# B&R Automation Studio project NAELD004C00R10L518F00 (part 40)

#### Act_Background_TCPSend.st
```iecst
(** 2021-08-01 **)
ACTION Act_Background_TCPSend:

	//Message Send (Generate XML Message)
	IF a_eMsgSend[0] <> HermesMsgTypeNA THEN

		IF a_eMsgSend[0] = HermesMsgTypeCheckAlive THEN
			fHermesFormCheckAlive(ADR(a_tyXMLTableDataSnd) , p_tyDTStructure , tyCheckAliveSnd);
			fTableConvertToXML(ADR(sSnd) , ADR(udiSndMsgLen) , SIZEOF(sSnd) , ADR(a_tyXMLTableDataSnd) , ADR(a_tyXMLTableDataSnd[0].sTitle) , ADR(a_tyXMLTableDataSnd[0].sValue) , ADR(a_tyXMLTableDataSnd[0].uiSize) , SIZEOF(a_tyXMLTableDataSnd[0]) , 12);

		ELSIF a_eMsgSend[0] = HermesMsgTypeCheckAlivePing THEN
			fHermesFormCheckAlive(ADR(a_tyXMLTableDataSnd) , p_tyDTStructure , tyCheckAlivePingSnd);
			fTableConvertToXML(ADR(sSnd) , ADR(udiSndMsgLen) , SIZEOF(sSnd) , ADR(a_tyXMLTableDataSnd) , ADR(a_tyXMLTableDataSnd[0].sTitle) , ADR(a_tyXMLTableDataSnd[0].sValue) , ADR(a_tyXMLTableDataSnd[0].uiSize) , SIZEOF(a_tyXMLTableDataSnd[0]) , 12);

		ELSIF a_eMsgSend[0] = HermesMsgTypeCheckAlivePong THEN
			fHermesFormCheckAlive(ADR(a_tyXMLTableDataSnd) , p_tyDTStructure , tyCheckAlivePongSnd);
			fTableConvertToXML(ADR(sSnd) , ADR(udiSndMsgLen) , SIZEOF(sSnd) , ADR(a_tyXMLTableDataSnd) , ADR(a_tyXMLTableDataSnd[0].sTitle) , ADR(a_tyXMLTableDataSnd[0].sValue) , ADR(a_tyXMLTableDataSnd[0].uiSize) , SIZEOF(a_tyXMLTableDataSnd[0]) , 12);

		ELSIF a_eMsgSend[0] = HermesMsgTypeServiceDescription THEN
			fHermesFormServiceDescription(ADR(a_tyXMLTableDataSnd) , p_tyDTStructure , tyServiceDescriptionSnd);
			fTableConvertToXML(ADR(sSnd) , ADR(udiSndMsgLen) , SIZEOF(sSnd) , ADR(a_tyXMLTableDataSnd) , ADR(a_tyXMLTableDataSnd[0].sTitle) , ADR(a_tyXMLTableDataSnd[0].sValue) , ADR(a_tyXMLTableDataSnd[0].uiSize) , SIZEOF(a_tyXMLTableDataSnd[0]) , 30);

		ELSIF a_eMsgSend[0] = HermesMsgTypeNotification THEN
			fHermesFormNotification(ADR(a_tyXMLTableDataSnd) , p_tyDTStructure , tyNotificationSnd);
			fTableConvertToXML(ADR(sSnd) , ADR(udiSndMsgLen) , SIZEOF(sSnd) , ADR(a_tyXMLTableDataSnd) , ADR(a_tyXMLTableDataSnd[0].sTitle) , ADR(a_tyXMLTableDataSnd[0].sValue) , ADR(a_tyXMLTableDataSnd[0].uiSize) , SIZEOF(a_tyXMLTableDataSnd[0]) , 14);

		ELSIF a_eMsgSend[0] = HermesMsgTypeBoardAvailable THEN
			fHermesFormBoardAvailable(ADR(a_tyXMLTableDataSnd) , p_tyDTStructure , tyBoardAvailableSnd);
			fTableConvertToXML(ADR(sSnd) , ADR(udiSndMsgLen) , SIZEOF(sSnd) , ADR(a_tyXMLTableDataSnd) , ADR(a_tyXMLTableDataSnd[0].sTitle) , ADR(a_tyXMLTableDataSnd[0].sValue) , ADR(a_tyXMLTableDataSnd[0].uiSize) , SIZEOF(a_tyXMLTableDataSnd[0]) , 50);

		ELSIF a_eMsgSend[0] = HermesMsgTypeRevokeBoardAvl THEN
			fHermesFormRevokeBoardAvailable(ADR(a_tyXMLTableDataSnd) , p_tyDTStructure);
			fTableConvertToXML(ADR(sSnd) , ADR(udiSndMsgLen) , SIZEOF(sSnd) , ADR(a_tyXMLTableDataSnd) , ADR(a_tyXMLTableDataSnd[0].sTitle) , ADR(a_tyXMLTableDataSnd[0].sValue) , ADR(a_tyXMLTableDataSnd[0].uiSize) , SIZEOF(a_tyXMLTableDataSnd[0]) , 8);

		ELSIF a_eMsgSend[0] = HermesMsgTypeMachineReady THEN
			eStatus1	:= Error;
			udiStatus1	:= 10135;	//Machine Ready Request To Send From Downstream Hermes

		ELSIF a_eMsgSend[0] = HermesMsgTypeRevokeMachineReady THEN
			eStatus1	:= Error;
			udiStatus1	:= 10136;	//Revoke Machine Ready Request To Send From Downstream Hermes

		ELSIF a_eMsgSend[0] = HermesMsgTypeStartTransport THEN
			eStatus1	:= Error;
			udiStatus1	:= 10137;	//Start Transport Request To Send From Downstream Hermes

		ELSIF a_eMsgSend[0] = HermesMsgTypeStopTransport THEN
			eStatus1	:= Error;
			udiStatus1	:= 10110;	//Stop Transport Request To Send From Downstream Hermes

		ELSIF a_eMsgSend[0] = HermesMsgTypeTransportFinished THEN
			fHermesFormTransportFinished(ADR(a_tyXMLTableDataSnd) , p_tyDTStructure , tyTransportFinished);
			fTableConvertToXML(ADR(sSnd) , ADR(udiSndMsgLen) , SIZEOF(sSnd) , ADR(a_tyXMLTableDataSnd) , ADR(a_tyXMLTableDataSnd[0].sTitle) , ADR(a_tyXMLTableDataSnd[0].sValue) , ADR(a_tyXMLTableDataSnd[0].uiSize) , SIZEOF(a_tyXMLTableDataSnd[0]) , 12);

		ELSIF a_eMsgSend[0] = HermesMsgTypeSetConfiguration THEN
			eStatus1	:= Error;
			udiStatus1	:= 10138;	//Set Configuration Request To Send From Downstream Hermes

		ELSIF a_eMsgSend[0] = HermesMsgTypeGetConfiguration THEN
			eStatus1	:= Error;
			udiStatus1	:= 10139;	//Get Configuration Request To Send From Downstream Hermes

		ELSIF a_eMsgSend[0] = HermesMsgTypeCurrConfiguration THEN
			eStatus1	:= Error;
			udiStatus1	:= 10140;	//Current Configuration Request To Send From Downstream Hermes

		ELSIF a_eMsgSend[0] = HermesMsgTypeBoardForecast THEN
			fHermesFormBoardForecast(ADR(a_tyXMLTableDataSnd) , p_tyDTStructure , tyBoardForecastSnd);
			fTableConvertToXML(ADR(sSnd) , ADR(udiSndMsgLen) , SIZEOF(sSnd) , ADR(a_tyXMLTableDataSnd) , ADR(a_tyXMLTableDataSnd[0].sTitle) , ADR(a_tyXMLTableDataSnd[0].sValue) , ADR(a_tyXMLTableDataSnd[0].uiSize) , SIZEOF(a_tyXMLTableDataSnd[0]) , 50);

		ELSIF a_eMsgSend[0] = HermesMsgTypeQueryBoardInfo THEN
			eStatus1	:= Error;
			udiStatus1	:= 10142;	//Query Board Info Request To Send From Downstream Hermes

		ELSIF a_eMsgSend[0] = HermesMsgTypeSendBoardInfo THEN
			fHermesFormSendBoardInfo(ADR(a_tyXMLTableDataSnd) , p_tyDTStructure , tySendBoardInfo);
			fTableConvertToXML(ADR(sSnd) , ADR(udiSndMsgLen) , SIZEOF(sSnd) , ADR(a_tyXMLTableDataSnd) , ADR(a_tyXMLTableDataSnd[0].sTitle) , ADR(a_tyXMLTableDataSnd[0].sValue) , ADR(a_tyXMLTableDataSnd[0].uiSize) , SIZEOF(a_tyXMLTableDataSnd[0]) , 40);
			bFoundTop	   := FALSE;
			bFoundBottom   := FALSE;
			bFoundNothing  := FALSE;
			bSearchTop     := FALSE;
			bSearchBottom  := FALSE;
			bSendOk        := FALSE;
			tyMsgTypeRcv.bQueryBoardInfo := FALSE;
			//10159

		ELSIF a_eMsgSend[0] = HermesMsgTypeQueryWorkOrderInfo THEN
			eStatus1	:= Error;
			udiStatus1	:= 10160;	//Query Work Order Info Request To Send From Downstream Hermes

		ELSIF a_eMsgSend[0] = HermesMsgTypeSendWorkOrderInfo THEN
			eStatus1	:= Error;
			udiStatus1	:= 10161;	//Send Work Order Info Request To Send From Downstream Hermes

		ELSIF a_eMsgSend[0] = HermesMsgTypeBoardArrived THEN
			eStatus1	:= Error;
			udiStatus1	:= 10162;	//BoardArrived Request To Send From Downstream Hermes

		ELSIF a_eMsgSend[0] = HermesMsgTypeBoardDeparted THEN
			eStatus1	:= Error;
			udiStatus1	:= 10163;	//BoardDeparted Request To Send From Downstream Hermes

		END_IF

		//Message Send
		IF p_bInternalUse = FALSE THEN
			fbSend.udiTCPIdent	:= udiClntIdent;
			fbSend.udiSndSize	:= udiSndMsgLen;
			fbSend(bEn := TRUE);
		ELSE
			sInternalSnd	:= sSnd;
		END_IF

		IF (fbSend.udiStatus = 0) OR (p_bInternalUse = TRUE) THEN

			fLogDTConvert(ADR(sDT) , p_dtCurrDT);
			memset(ADR(a_sLogList[udiLogCntr]) , 0 , SIZEOF(a_sLogList[udiLogCntr]));
			memcpy(ADR(a_sLogList[udiLogCntr]) + LEN(a_sLogList[udiLogCntr]) , ADR(sDT) , LEN(sDT));
			memcpy(ADR(a_sLogList[udiLogCntr]) + LEN(a_sLogList[udiLogCntr]) , ADR('$r$n') , LEN('$r$n'));
			memcpy(ADR(a_sLogList[udiLogCntr]) + LEN(a_sLogList[udiLogCntr]) , ADR('SND_TO_DS$r$n') , LEN('SND_TO_DS$r$n'));
			memcpy(ADR(a_sLogList[udiLogCntr]) + LEN(a_sLogList[udiLogCntr]) , ADR(sSnd) , LEN(sSnd));
			memcpy(ADR(a_sLogList[udiLogCntr]) + LEN(a_sLogList[udiLogCntr]) , ADR('$r$n$r$n') , LEN('$r$n$r$n'));

			udiLogCntr	:= udiLogCntr + 1;
			IF udiLogCntr = 11 THEN
				udiLogCntr	:= 1;
			END_IF

			Act_Background_NotificationSnd;
			fHermesRmvOneMsgSend(ADR(a_eMsgSend) , ADR(udiMsgSendBffr));

			fbSend(bEn := FALSE);

		ELSIF (fbSend.udiStatus = 2321) AND (p_bInternalUse = FALSE) THEN
			bRstConnection	:= TRUE;

		ELSIF (fbSend.udiStatus < 65534) AND (p_bInternalUse = FALSE) THEN
			eStatus1	:= Error;

			IF fbSend.udiStatus = 2300 THEN
				udiStatus1	:= 10143;	//Invalid Ident While Sending Data
			ELSIF fbSend.udiStatus = 2320 THEN
				udiStatus1	:= 10144;	//TCP Retry Send Data Error While Sending Data
			ELSIF fbSend.udiStatus = 2322 THEN
				udiStatus1	:= 10145;	//TCP Send Data Error
			ELSE
				udiStatus1	:= fbSend.udiStatus;
			END_IF

		END_IF

	END_IF

END_ACTION
```

#### Act_InitGlobal.st
```iecst
(** 2019-03-25 **)
ACTION Act_InitGlobal:

	(* Always Change If Project Change *)

	//Pass Data To Link
	p_bLinkStartupRun ACCESS p_StartupRun;
	p_eLinkMcParamDSCommMod ACCESS p_McParamDSCommAMod;

	p_usiLinkProdRcpCurrRcpFlipBrd ACCESS p_ProdRcpCurrRcp2FlippedBrd;
	p_bLinkConvHvBrd ACCESS p_PullConvHvBrd;
	p_bLinkOpsTravLifLDDSComm ACCESS p_OpsTravLifLDDSComm;
	p_eLinkTravLifLDPosGo ACCESS p_OpsTravLifLDPosGo;

	//Pass Data To Internal Use
	p_udiRstErr ACCESS p_RstErrReset;
	p_bPrep ACCESS p_NtParamHermesPrep;
	p_tyParam ACCESS p_HermesDSParam1;
	p_sIPAddr ACCESS p_HWInfoIPAddr;
	pa_usiMacAddr ACCESS p_HWInfoMacAddr;
	p_tyDTStructure ACCESS p_TimeCurrDTStruct;
	p_dtCurrDT ACCESS p_TimeCurrDT;
	p_sMcId ACCESS p_McParamMcNm;
	p_sRecipeNm ACCESS p_ProdRcpCurrRcp1Nm;
	p_sWorkOrderId ACCESS p_AutoRcpWorkOrderId; //from autorcp /////////p_SvyHermesWorkOrderId; //Work Order Id from SupervisoryHermes
	p_sBatchId ACCESS p_SvyHermesBatchId; //Batch Id from SupervisoryHermes
	p_diWidthInUM ACCESS p_ProdRcpCurrRcp1Width;
	p_udiAliveIdleTimeInSec ACCESS p_NtParamDSHermesAAliveTmInSec;
	p_tConnTimeOut ACCESS p_NtParamDSHermesAConnTO;
	p_diTransferInTO ACCESS p_McParamTranOutErrDlyTm;
	pa_tyXMLTableDataBrdAvl ACCESS p_HermesBrdAvlDataTableLastZ; //Last zone Board Data, for B.A
	p_iXMLTableDataBrdAvlTtlIdx ACCESS p_HermesBrdAvlDataTtlIdxLastZ;  //Last zone Board Data, for B.A
	p_bNewBrdAvlFirstZone ACCESS p_HermesBrdAvlDataNewBrdAvl1stZ; //First zone Board Data, for B.F
	p_bNewBrdAvlLastZone ACCESS p_HermesBrdAvlDataNewBrdAvlLastZ; //Last zone Board Data, for B.A
	p_bOpsRun ACCESS p_OpsRun;
	p_bInterruptSen ACCESS p_DIConvRgtSen; //Last Zone Sensor that give B.A
	p_udiFileKeepDay ACCESS p_NtParamDSHermesAFileKeepDay;
	p_sRetainFileName ACCESS p_NtParamDSHermesRetainFileNm;
	p_sProgNm ACCESS p_NtParamDSHermesAProgNm;
	p_bNtSettingsLoadDone ACCESS p_StartupNtSettingsLoadDone;
	p_bRmtPrep ACCESS p_NtParamHermesRmtPrep;
	p_bRmtEn ACCESS p_McParamHermesRmtEn;
	p_bSvyPrep ACCESS p_NtParamHermesSvyPrep;
	p_bSvyEn ACCESS p_McParamHermesSvyEn;
	p_bOpsGConv1HvBrd ACCESS p_PullConvHvBrd; //Take Zone 1's Have Board
	//p_tyUSBoardArrivedData ACCESS p_USHermesBoardArrivedData;
	//p_rAWCycleTm ACCESS p_NtParamDSHermesAWCycleTm;
	p_bInitDone ACCESS p_OpsTravLifLDInitDone;
	p_bFirstZoneEndSen ACCESS p_DIConvRgtSen; //Take First Zone's End sensor
	p_tyHermesConfiguration ACCESS p_HermesConfiguration;
//	p_bUSHermesStopTransport ACCESS p_USHermesStopTransportSnd;
//	p_bRcvBoardInfo ACCESS p_USHermesRcvBoardInfoOk;
//	p_tyBoardInfoData ACCESS p_USHermesBoardInfoData; //SendBoardInfo from Upstream, used to generate B.A for inserted PCB
//	p_bUSHermesTransporting ACCESS p_USHermesTransporting;
	p_eLinkCustomerReq ACCESS p_NtParamCustomerReq;
	p_usiProdRcpCurrRcp1McMod  ACCESS  p_ProdRcpCurrRcp1McMod;      //ADD
//	p_usiSelProdRcpStep  ACCESS p_SelProdRcpStep;

	// phase 1
	p_tySendWorkOrderData ACCESS p_SvyHermesSendWorkOrderData;
	p_bReplyWorkOrderInfo ACCESS  p_ReplyWorkOrderInfo;
	p_bSendBoardForecast ACCESS p_SendBoardForecast;
	p_bClearWorkOrder ACCESS p_ClearWorkOrder;

	p_tyAutoRcpTravLif ACCESS p_AutoRcpTravLif;
	p_diLinkAutoRcpTravLifWidth ACCESS p_AutoRcpTravLifWidth;
	p_diLinkAutoRcpMag1Width ACCESS p_diAutoRcpMag1Width;
	p_diLinkAutoRcpMag2Width ACCESS p_diAutoRcpMag2Width;
	p_diLinkAutoRcpMag3Width ACCESS p_diAutoRcpMag3Width;

	p_tyAutoRcpMagRcp ACCESS p_AutoRcpMagRcp;
	p_ausiSvyMagAccOrder ACCESS p_SvyHermesMagAccOrder;

	p_sHermesBrdId ACCESS p_HermesBrdId;
	p_bDIPullerRetRS ACCESS p_DIPullerRetRS;
	(* Always Change If Project Change *)
END_ACTION
```

#### Act_Initial.st
```iecst
(** 2021-08-01 **)
ACTION Act_Initial:

	//Initial
	sStatTxt	:= a_sStatText[eStat];

	fbCreateSvr.udiSndBffrSize		:= p_udiSndBffrSize;
	fbCreateSvr.udiRcvBffrSize		:= p_udiRcvBffrSize;
	fbCreateSvr.udiAliveIdleTmInSec	:= p_udiAliveIdleTimeInSec;
	fbCreateSvr(bEn := FALSE);

	fbListen(bEn := FALSE);

	fbRcv.udiBffrSize	:= SIZEOF(sRcv);
	fbRcv.p_BffrDest	:= ADR(sRcv);
	fbRcv(bEn := FALSE);

	fbSend.p_BffrDest	:= ADR(sSnd);
	fbSend(bEn := FALSE);

	fbCloseSvr(bEn := FALSE);
	fbCloseClnt(bEn := FALSE);

	fbParseXMLTable.p_XMLTable	:= ADR(a_tyXMLTableDataRcv);

	fbCheckAlive(bEn := FALSE);

	fbCheckAliveSendPing(bEn := FALSE);

	fbCheckAliveRcvPing(bEn := FALSE);

	fbSequenceDS.p_tyMsgTypeRcv	:= ADR(tyMsgTypeRcv);
	fbSequenceDS(bEn := FALSE);

	fbSequenceTO(bEn := FALSE);

	fbFileAppend1.sDevice	:= 'Log';
	fbFileAppend1(bEn := FALSE);

	fbFileOldDel1.sDevice			:= 'Log';
	fbFileOldDel1.sPath				:= '';
	fbFileOldDel1.sKeyword			:= p_sProgNm;
	fbFileOldDel1.udiFileKeepDay	:= p_udiFileKeepDay;
	fbFileOldDel1(bEn := FALSE);

	fbFileRead1.sDevice			:= 'Retain';
	fbFileRead1.sFile			:= p_sRetainFileName;
	fbFileRead1.udiOffset		:= 0;
	fbFileRead1(bEn := FALSE);

	fbFileWrite1.sDevice		:= 'Retain';
	fbFileWrite1.sFile			:= p_sRetainFileName;
	fbFileWrite1.udiOffset		:= 0;
	fbFileWrite1.udiOption		:= 0;
	fbFileWrite1(bEn := FALSE);

END_ACTION
```

#### Act_InitLocal.st
```iecst
(** 2021-08-01 **)
ACTION Act_InitLocal:

	//Input Reference Link To Local Variable
	p_eAct ACCESS ADR(eAct);
	p_udiRstErr ACCESS ADR(udiRstErr);
	p_bPrep ACCESS ADR(bPrep);
	p_bEn ACCESS ADR(bEn);
	p_bDis ACCESS ADR(bDis);
	p_tyParam ACCESS ADR(tyParam);
	p_sIPAddr ACCESS ADR(sIPAddr);
	pa_usiMacAddr ACCESS ADR(a_usiMacAddr);
	p_tyDTStructure ACCESS ADR(tyDTStructure);
	p_dtCurrDT ACCESS ADR(dtCurrDT);
	p_bRdySnd ACCESS ADR(bRdySnd);
	p_bSndCompl ACCESS ADR(bSndCompl);
	p_bSndIncompl ACCESS ADR(bSndInCompl);
	p_bSndNotStart ACCESS ADR(bSndNotStart);
	p_bBAWidthEn ACCESS ADR(bBAWidthEn);
	p_bBASltEn ACCESS ADR(bBASltEn);
	p_bBFWidthEn ACCESS ADR(bBFWidthEn);
	p_bBFSltEn ACCESS ADR(bBFSltEn);
	p_sForecastId ACCESS ADR(sForecastId);
	p_sBoardId ACCESS ADR(sBoardId);
	p_sMcId ACCESS ADR(sMcId);
	p_sInterfaceId ACCESS ADR(sInterfaceId);
	p_sVersion ACCESS ADR(sVersion);
	p_eFailedBoard ACCESS ADR(eFailedBoard);
	p_sRecipeNm ACCESS ADR(sRecipeNm);
	p_eFlippedBoard ACCESS ADR(eFlippedBoard);
	p_sTopBarcode ACCESS ADR(sTopBarcode);
	p_sBottomBarcode ACCESS ADR(sBottomBarcode);
	p_rLength ACCESS ADR(rLength);
	p_rThickness ACCESS ADR(rThickness);
	p_rConveyorSpeed ACCESS ADR(rConveyorSpeed);
	p_rTopClearanceHeight ACCESS ADR(rTopClearanceHeight);
	p_rBottomClearanceHeight ACCESS ADR(rBottomClearanceHeight);
	p_rWeight ACCESS ADR(rWeight);
	p_sWorkOrderId ACCESS ADR(sWorkOrderId);
	p_sBatchId ACCESS ADR(sBatchId);
	p_diWidthInUM ACCESS ADR(diWidthInUM);
	p_diMinSltValue ACCESS ADR(diMinSltValue);
	p_diMaxSltValue ACCESS ADR(diMaxSltValue);
	p_diPitch ACCESS ADR(diPitch);
	p_diTtlSlt ACCESS ADR(diTtlSlt);
	p_diSltToSltInUM ACCESS ADR(diSltToSltInUM);
	p_udiSndBffrSize ACCESS ADR(udiSndBffrSize);
	p_udiRcvBffrSize ACCESS ADR(udiRcvBffrSize);
	p_udiAliveIdleTimeInSec ACCESS ADR(udiAliveIdleTimeInSec);
	p_tConnTimeOut ACCESS ADR(tConnTimeOut);
	p_diTransferInTO ACCESS ADR(diTransferInTO);
	pa_tyXMLTableDataBrdAvl ACCESS ADR(a_tyXMLTableDataBrdAvl);
	p_iXMLTableDataBrdAvlTtlIdx ACCESS ADR(iXMLTableDataBrdAvlTtlIdx);
	p_bNewBrdAvlFirstZone ACCESS ADR(bNewBrdAvl1);
	p_bNewBrdAvlLastZone ACCESS ADR(bNewBrdAvl2);
	p_bOpsRun ACCESS ADR(bOpsRun);
	p_bInterruptSen ACCESS ADR(bInterruptSen);
	p_udiFileKeepDay ACCESS ADR(udiFileKeepDay);
	p_sRetainFileName ACCESS ADR(sRetainFileName);
	p_udiRetainDataAddr ACCESS ADR(udiRetainDataAddr);
	p_udiRetainDataLen ACCESS ADR(udiRetainDataLen);
	p_sProgNm ACCESS ADR(sProgNm);
	p_bNtSettingsLoadDone ACCESS ADR(bNtSettingsLoadDone);
	p_bRmtPrep ACCESS ADR(bRmtPrep);
	p_bRmtEn ACCESS ADR(bRmtEn);
	p_bSvyPrep ACCESS ADR(bSvyPrep);
	p_bSvyEn ACCESS ADR(bSvyEn);
	p_bOpsGConv1HvBrd ACCESS ADR(bOpsGConv1HvBrd);
	p_tyUSBoardArrivedData ACCESS ADR(tyUSBoardArrivedData);
	p_rMcCycleTm ACCESS ADR(rMachineCycleTime);
	p_rAWCycleTm ACCESS ADR(rAutoWidthCycleTime);
	p_bInitDone ACCESS ADR(bInitDone);
	p_bFirstZoneEndSen ACCESS ADR(bFirstZoneEndSen);
	p_bFirstZoneHaveBoard ACCESS ADR(bFirstZoneHaveBoard);
	p_bNewProduct ACCESS ADR(bNewProduct);
	p_bNewWidth ACCESS ADR(bNewWidth);
	p_tyHermesConfiguration ACCESS ADR(tyHermesCurrConfiguration);
	p_bUSHermesStopTransport ACCESS ADR(bUSHermesStopTransport);
	p_bRcvBoardInfo ACCESS ADR(bRcvBoardInfo);
	p_tyBoardInfoData ACCESS ADR(tyBoardInfoData);
	p_bUSHermesTransporting ACCESS ADR(bUSHermesTransporting);
	p_bInternalUse ACCESS ADR(bInternalUse);
	p_sInternalRcv ACCESS ADR(sInternalRcv);

END_ACTION
```

#### Act_Link.st
```iecst
(** 2021-08-01 **)
ACTION Act_Link:

	//Receive Alive Time
	p_tyParam.tRcvAlive	:= p_tyParam.tSndAlive * 2;

	//Ready Send
	//Transfer Finished
//	IF (p_eLinkConvDir = ConvDirLToR) OR (p_eLinkConvDir = ConvDirRToR) THEN
		IF EDGENEG(p_bFirstZoneEndSen) THEN
			p_bSndCompl	:= TRUE;
		END_IF
//	ELSE
//		IF EDGENEG(p_bLinkDILeftSen) THEN
//			p_bSndCompl	:= TRUE;
//		END_IF
//	END_IF

	//Good Bad Board
//	IF p_bLinkOpsConvGdBrd = TRUE THEN
		p_eFailedBoard	:= HermesGoodBoard;
//	ELSE
//		p_eFailedBoard	:= HermesFailedBoard;
//	END_IF

	//New Product for Board Forecast(Id)
	//p_bNewProduct will be True only when machine accepted new recipe, can perform ChangeOver, i.e Machine Free (all zones).
		//siemen
	IF p_ausiSvyMagAccOrder[1] = 10 AND p_bDIPullerRetRS THEN
		p_bNewProduct := (p_tyAutoRcpTravLif.sWorkOrderId <> p_tyAutoRcpMagRcp[1].sWorkOrderId OR
						p_tyAutoRcpTravLif.sProductTypeId <> p_tyAutoRcpMagRcp[1].sProductTypeId OR
						p_tyAutoRcpTravLif.sBatchId <> p_tyAutoRcpMagRcp[1].sBatchId OR
						p_tyAutoRcpTravLif.rWidth <> p_tyAutoRcpMagRcp[1].rWidth) AND (p_bLinkStartupRun = FALSE);
	ELSIF p_ausiSvyMagAccOrder[2] = 10 AND p_bDIPullerRetRS THEN
		p_bNewProduct := (p_tyAutoRcpTravLif.sWorkOrderId <> p_tyAutoRcpMagRcp[2].sWorkOrderId OR
						p_tyAutoRcpTravLif.sProductTypeId <> p_tyAutoRcpMagRcp[2].sProductTypeId OR
						p_tyAutoRcpTravLif.sBatchId <> p_tyAutoRcpMagRcp[2].sBatchId OR
						p_tyAutoRcpTravLif.rWidth <> p_tyAutoRcpMagRcp[2].rWidth) AND (p_bLinkStartupRun = FALSE);
	ELSIF p_ausiSvyMagAccOrder[3] = 10 AND p_bDIPullerRetRS THEN
		p_bNewProduct := (p_tyAutoRcpTravLif.sWorkOrderId <> p_tyAutoRcpMagRcp[3].sWorkOrderId OR
						p_tyAutoRcpTravLif.sProductTypeId <> p_tyAutoRcpMagRcp[3].sProductTypeId OR
						p_tyAutoRcpTravLif.sBatchId <> p_tyAutoRcpMagRcp[3].sBatchId OR
						p_tyAutoRcpTravLif.rWidth <> p_tyAutoRcpMagRcp[3].rWidth) AND (p_bLinkStartupRun = FALSE);
	ELSE
		p_bNewProduct := FALSE;
	END_IF

	//p_bNewProduct := ((*(EDGEPOS(p_bLinkProdRcpCurrAll[0].sRcpNm = p_bLinkProdRcpCurrAll[1].sRcpNm)*)) AND (p_bLinkStartupRun = FALSE));
	bBFAccNewWidth[1] :=  p_diLinkAutoRcpTravLifWidth = p_diLinkAutoRcpMag1Width AND p_eLinkTravLifLDPosGo = TravLifLDPosUS1;
	bBFAccNewWidth[2] :=	p_diLinkAutoRcpTravLifWidth = p_diLinkAutoRcpMag2Width AND p_eLinkTravLifLDPosGo = TravLifLDPosUS2;
	bBFAccNewWidth[3] :=	p_diLinkAutoRcpTravLifWidth = p_diLinkAutoRcpMag3Width AND p_eLinkTravLifLDPosGo = TravLifLDPosUS3;
	//p_bNewWidth will be True only when machine accepted new width, can perform ChangeOver, i.e Machine Free (all zones).
	//p_bNewWidth :=   (EDGEPOS(bBFAccNewWidth[1]) OR EDGEPOS(bBFAccNewWidth[2]) OR EDGEPOS(bBFAccNewWidth[3])) AND (p_bLinkStartupRun = FALSE);

	p_bRdySnd	:= p_bLinkOpsTravLifLDDSComm AND p_eLinkTravLifLDPosGo = TravLifLDPosDS1;  //DBA

	//Machine Cycle Time
	p_rMcCycleTm ACCESS p_NtParamDSHermesMcCycleTm; //Change this if machine got Worst/Least/Different Cycle Time accordingly

	//Flipped Board
	p_eFlippedBoard	:= USINT_TO_UDINT(p_usiLinkProdRcpCurrRcpFlipBrd);

	//Machine All Empty(for ChangeOver), adjust accordingly                                                            //Add
	bAllZonesEmpty := p_bOpsGConv1HvBrd = FALSE AND p_bFirstZoneEndSen = FALSE;// AND p_bLinkDIPresentSen = FALSE (*AND p_tyDI.bTopCoverSWSig = TRUE*);

	//Machine First Zone have board
	p_bFirstZoneHaveBoard := (p_bUSHermesStopTransport AND p_bOpsGConv1HvBrd) OR (p_bOpsGConv1HvBrd AND p_bUSHermesTransporting = FALSE); //Zone 1 have board, either PCB_In from upstream Or Manually load PCB at Zone 1

END_ACTION
```

#### Act_LinkAction.st
```iecst
(** 2021-08-01 **)
ACTION Act_LinkAction:

	IF p_bLinkStartupRun = TRUE THEN
		p_eAct ACCESS p_StartupDSHermesAAct;
	ELSE
		p_eAct ACCESS ADR(eAct);

		IF EDGEPOS(p_eLinkMcParamDSCommMod = McSetCommModHermes) THEN
			bHermesRun	:= TRUE;
			bHermesStop	:= FALSE;
		END_IF

		IF EDGENEG(p_eLinkMcParamDSCommMod = McSetCommModHermes) THEN
			bHermesRun	:= FALSE;
			bHermesStop	:= TRUE;
		END_IF

		IF bHermesRun = TRUE THEN
			p_eAct	:= HermesActBGStartRun;

			IF (eStat = HermesActBGStartRun) AND (eStatus = Done) THEN
				p_eAct		:= HermesActIdle;
				bHermesRun	:= FALSE;
			END_IF
		END_IF

		IF bHermesStop = TRUE THEN
			p_eAct	:= HermesActBGStopRun;

			IF (eStat = HermesActBGStopRun) AND (eStatus = Done) THEN
				p_eAct		:= HermesActIdle;
				bHermesStop	:= FALSE;
			END_IF
		END_IF

	END_IF

//Delete Old Log File for 24 hours After Machine is Continuous Running 30 Days.

	fbDlyTmr(IN := TRUE);
	IF fbDlyTmr.Q THEN
		fbDeleteLogTmr (IN := TRUE);
		IF fbDeleteLogTmr.Q AND eStatus <> Busy THEN
			p_eAct := HermesActDeleteOldLog;
			IF eStat = HermesActDeleteOldLog AND eStatus = Done THEN
				p_eAct := HermesActIdle;
				fbDlyTmr (IN := FALSE);
				fbDeleteLogTmr (IN := FALSE);
			END_IF
		END_IF
	END_IF
END_ACTION
```

#### Cyclic.st
```iecst
(** 2021-08-01 **)
PROGRAM _CYCLIC

	IF bInitDone = FALSE THEN
		bInitDone	:= TRUE;

		Act_InitLocal;
		Act_InitGlobal;

	ELSIF bInitialDone = FALSE THEN
		IF p_bNtSettingsLoadDone = TRUE THEN
			bInitialDone	:= TRUE;

			Act_Initial;
		END_IF

	ELSE

		Act_RstErr;
		Act_LinkAction;
		Act_Action;
		Act_LinkEn;

		IF (p_bPrep = TRUE) AND (p_bEn = TRUE) AND (p_bDis = FALSE) THEN
			Act_Link;
			Act_Main;
			Act_Background;
			Act_Background_ProcessData;
		ELSE
			Act_Main_Disable;

			IF eStat <> HermesActIdle THEN
				eStatus	:= Done;
			ELSE
				eStatus	:= Idle;
			END_IF
		END_IF

		Act_CombineErr;
		Act_Alarm;
		Act_Alarm1;
		Act_Alarm2;
		Act_Alarm3;
		Act_Alarm4;
	END_IF

END_PROGRAM
```

#### Init.st
```iecst
(** 2021-08-01 **)
PROGRAM _INIT

	(* Always Change If Project Change *)

	//Pass Address To Global Address For External Use
	//Action, State & Status
	p_DSHermesAStat	    	:= ADR(eStat);
	p_DSHermesAStatus    	:= ADR(eMainStatus);
	p_DSHermesAStatTxt    	:= ADR(sStatTxt);

	//Alarm
	p_DSHermesAAlmData    	:= ADR(tyAlmData);
	p_DSHermesAAlmData1	    := ADR(tyAlmData1);
	p_DSHermesAAlmData2    	:= ADR(tyAlmData2);
	p_DSHermesAAlmData3    	:= ADR(tyAlmData3);
	p_DSHermesAAlmData4    	:= ADR(tyAlmData4);//add

	//Output
	p_DSHermesAFileNotFound		    := ADR(bFileNotFound);
	p_DSHermesAConnected		    := ADR(bConnected);
	p_DSHermesAHandshakeDone	    := ADR(bHandshakeDone);
	p_DSHermesAUSRdy			    := ADR(bUSRdy);
	p_DSHermesADSRdy			    := ADR(bDSRdy);
	p_DSHermesAUSGdRdy		    	:= ADR(bUSGdRdy);
	p_DSHermesADSGdRdy		    	:= ADR(bDSGdRdy);
	p_DSHermesATransporting	    	:= ADR(bTransporting);
	p_DSHermesAStopTransport	    := ADR(bStopTransport);
	p_DSHermesAInternalSnd	    	:= ADR(sInternalSnd);
	p_DSHermesATransportFinishedSnd  := ADR(bTransportFinishedSnd);
	p_DSHermesABoardDepartedData     := ADR(tyBoardDepartedInfo);
	p_DSHermesAAllZonesEmpty         := ADR(bAllZonesEmpty);

	p_SendBFId                     := ADR (bSendBFId);        //ADD

	(* Always Change If Project Change *)

END_PROGRAM
```

### DSHermesB.var - Change By Project
```iecst
(*2021-08-01*)
(**)
(*Action & State & Status*)
VAR
	p_DSHermesBStat : UDINT;
	p_DSHermesBStatus : UDINT;
	p_DSHermesBStatTxt : UDINT;
END_VAR
(**)
(*Alarm*)
VAR
	p_DSHermesBAlmData : UDINT;
	p_DSHermesBAlmData1 : UDINT;
	p_DSHermesBAlmData2 : UDINT;
	p_DSHermesBAlmData3 : UDINT;
	p_DSHermesBAlmData4 : UDINT;
END_VAR
(**)
(*Output*)
VAR
	p_DSHermesBFileNotFound : UDINT;
	p_DSHermesBConnected : UDINT;
	p_DSHermesBHandshakeDone : UDINT;
	p_DSHermesBUSRdy : UDINT;
	p_DSHermesBDSRdy : UDINT;
	p_DSHermesBUSGdRdy : UDINT;
	p_DSHermesBDSGdRdy : UDINT;
	p_DSHermesBTransporting : UDINT;
	p_DSHermesBStopTransport : UDINT;
	p_DSHermesBInternalSnd : UDINT;
	p_DSHermesBTransportFinishedSnd : UDINT;
	p_DSHermesBBoardDepartedData : UDINT;
	p_DSHermesBAllZonesEmpty : UDINT;
	p_SendBFIdB : UDINT;
END_VAR
```

### Program Logical/Hermes/DSHermesB (IEC, version 1.00.0) - 1.00.0 - NtHermes v5.00.0 , NtTCP v5.00.0 , NtMessage v5.00.0

#### Init.st - Change By Project
```iecst
(** 2021-08-01 **)
PROGRAM _INIT

	(* Always Change If Project Change *)

	//Pass Address To Global Address For External Use
	//Action, State & Status
	p_DSHermesBStat	    	:= ADR(eStat);
	p_DSHermesBStatus    	:= ADR(eMainStatus);
	p_DSHermesBStatTxt    	:= ADR(sStatTxt);

	//Alarm
	p_DSHermesBAlmData    	:= ADR(tyAlmData);
	p_DSHermesBAlmData1	    := ADR(tyAlmData1);
	p_DSHermesBAlmData2    	:= ADR(tyAlmData2);
	p_DSHermesBAlmData3    	:= ADR(tyAlmData3);
	p_DSHermesBAlmData4    	:= ADR(tyAlmData4);//add

	//Output
	p_DSHermesBFileNotFound		    := ADR(bFileNotFound);
	p_DSHermesBConnected		    	:= ADR(bConnected);
	p_DSHermesBHandshakeDone	    	:= ADR(bHandshakeDone);
	p_DSHermesBUSRdy			    	:= ADR(bUSRdy);
	p_DSHermesBDSRdy			    	:= ADR(bDSRdy);
	p_DSHermesBUSGdRdy		    	:= ADR(bUSGdRdy);
	p_DSHermesBDSGdRdy		    	:= ADR(bDSGdRdy);
	p_DSHermesBTransporting	    	:= ADR(bTransporting);
	p_DSHermesBStopTransport	    	:= ADR(bStopTransport);
	p_DSHermesBInternalSnd	    	:= ADR(sInternalSnd);
	p_DSHermesBTransportFinishedSnd  := ADR(bTransportFinishedSnd);
	p_DSHermesBBoardDepartedData     := ADR(tyBoardDepartedInfo);
	p_DSHermesBAllZonesEmpty         := ADR(bAllZonesEmpty);

	p_SendBFIdB                     := ADR (bSendBFId);        //ADD

	(* Always Change If Project Change *)

END_PROGRAM
```

#### Act_InitGlobal.st - Change By Project
```iecst
(** 2019-03-25 **)
ACTION Act_InitGlobal:

	(* Always Change If Project Change *)

	//Pass Data To Link
	p_bLinkStartupRun ACCESS p_StartupRun;
	p_eLinkMcParamDSCommMod ACCESS p_McParamDSCommBMod;
	p_bLinkNtParamProjLaneBPrep ACCESS p_NtParamProjLaneBPrep;

	p_usiLinkProdRcpCurrRcpFlipBrd ACCESS p_ProdRcpCurrRcp2FlippedBrd;
	p_bLinkConvHvBrd ACCESS p_PullConvHvBrd;
	p_bLinkOpsTravLifLDDSComm ACCESS p_OpsTravLifLDDSComm;
	p_eLinkTravLifLDPosGo ACCESS p_OpsTravLifLDPosGo;

	//Pass Data To Internal Use
	p_udiRstErr ACCESS p_RstErrReset;
	p_bPrep ACCESS p_NtParamHermesPrep;
	p_tyParam ACCESS p_HermesDSParam2;
	p_sIPAddr ACCESS p_HWInfoIPAddr;
	pa_usiMacAddr ACCESS p_HWInfoMacAddr;
	p_tyDTStructure ACCESS p_TimeCurrDTStruct;
	p_dtCurrDT ACCESS p_TimeCurrDT;
	p_sMcId ACCESS p_McParamMcNm;
	p_sRecipeNm ACCESS p_ProdRcpCurrRcp1Nm;
	p_sWorkOrderId ACCESS p_SvyHermesWorkOrderId; //Work Order Id from SupervisoryHermes
	p_sBatchId ACCESS p_SvyHermesBatchId; //Batch Id from SupervisoryHermes
	p_diWidthInUM ACCESS p_ProdRcpCurrRcp1Width;
	p_udiAliveIdleTimeInSec ACCESS p_NtParamDSHermesBAliveTmInSec;
	p_tConnTimeOut ACCESS p_NtParamDSHermesBConnTO;
	p_diTransferInTO ACCESS p_McParamTranOutErrDlyTm;
	pa_tyXMLTableDataBrdAvl ACCESS p_HermesBrdAvlDataTableLastZ; //Last zone Board Data, for B.A
	p_iXMLTableDataBrdAvlTtlIdx ACCESS p_HermesBrdAvlDataTtlIdxLastZ;  //Last zone Board Data, for B.A
	p_bNewBrdAvlFirstZone ACCESS p_HermesBrdAvlDataNewBrdAvl1stZ; //First zone Board Data, for B.F
	p_bNewBrdAvlLastZone ACCESS p_HermesBrdAvlDataNewBrdAvlLastZ; //Last zone Board Data, for B.A
	p_bOpsRun ACCESS p_OpsRun;
	p_bInterruptSen ACCESS p_DIConvRgtSen; //Last Zone Sensor that give B.A
	p_udiFileKeepDay ACCESS p_NtParamDSHermesBFileKeepDay;
	p_sRetainFileName ACCESS p_NtParamDSHermesRetainFileNm;
	p_sProgNm ACCESS p_NtParamDSHermesBProgNm;
	p_bNtSettingsLoadDone ACCESS p_StartupNtSettingsLoadDone;
	p_bRmtPrep ACCESS p_NtParamHermesRmtPrep;
	p_bRmtEn ACCESS p_McParamHermesRmtEn;
	p_bSvyPrep ACCESS p_NtParamHermesSvyPrep;
	p_bSvyEn ACCESS p_McParamHermesSvyEn;
	p_bOpsGConv1HvBrd ACCESS p_PullConvHvBrd; //Take Zone 1's Have Board
//	p_tyUSBoardArrivedData ACCESS p_USHermesBoardArrivedData;
//	p_rAWCycleTm ACCESS p_NtParamDSHermesAWCycleTm;
	p_bInitDone ACCESS p_OpsTravLifLDInitDone;
	p_bFirstZoneEndSen ACCESS p_DIConvRgtSen; //Take First Zone's End sensor
	p_tyHermesConfiguration ACCESS p_HermesConfiguration;
//	p_bUSHermesStopTransport ACCESS p_USHermesStopTransportSnd;
//	p_bRcvBoardInfo ACCESS p_USHermesRcvBoardInfoOk;
//	p_tyBoardInfoData ACCESS p_USHermesBoardInfoData; //SendBoardInfo from Upstream, used to generate B.A for inserted PCB
//	p_bUSHermesTransporting ACCESS p_USHermesTransporting;
	p_eLinkCustomerReq ACCESS p_NtParamCustomerReq;
	p_usiProdRcpCurrRcp1McMod  ACCESS  p_ProdRcpCurrRcp1McMod;      //ADD
//	p_usiSelProdRcpStep  ACCESS p_SelProdRcpStep;

	// phase 1
	p_tySendWorkOrderData ACCESS p_SvyHermesSendWorkOrderData;
	p_bReplyWorkOrderInfo ACCESS  p_ReplyWorkOrderInfo;
	p_bSendBoardForecast ACCESS p_SendBoardForecast;
	p_bClearWorkOrder ACCESS p_ClearWorkOrder;

	(* Always Change If Project Change *)
END_ACTION
```

#### InputRef_Link.var - Change By Project
```iecst
(*2021-08-01*)
(**)
VAR
	p_bLinkAWWidthPosDiff : REFERENCE TO BOOL;
	p_bLinkOpsAWStepMove : REFERENCE TO BOOL;
	p_bLinkProdRcpCurrAll : REFERENCE TO ARRAY[0..5] OF tyProdRcpParam;
END_VAR
(**)
VAR
	p_bLinkStartupRun : REFERENCE TO BOOL;
	p_eLinkMcParamDSCommMod : REFERENCE TO eMcSetCommMod;
	p_bLinkNtParamProjLaneBPrep : REFERENCE TO BOOL;
	bHermesRun : BOOL;
	bHermesStop : BOOL;
END_VAR
(**)
VAR
	p_usiLinkProdRcpCurrRcpFlipBrd : REFERENCE TO USINT;
	p_bLinkConvHvBrd : REFERENCE TO BOOL;
	p_bLinkOpsTravLifLDDSComm : REFERENCE TO BOOL;
	p_eLinkTravLifLDPosGo : REFERENCE TO eTravLifLDPos;
	p_eLinkCustomerReq : REFERENCE TO eCustomer;
END_VAR
```

#### Act_LinkAction.st - Change By Project
```iecst
(** 2021-08-01 **)
ACTION Act_LinkAction:

	IF p_bLinkStartupRun = TRUE THEN
		p_eAct ACCESS p_StartupDSHermesBAct;
	ELSE
		p_eAct ACCESS ADR(eAct);

		IF EDGEPOS(p_eLinkMcParamDSCommMod = McSetCommModHermes) THEN
			bHermesRun	:= TRUE;
			bHermesStop	:= FALSE;
		END_IF

		IF EDGENEG(p_eLinkMcParamDSCommMod = McSetCommModHermes) THEN
			bHermesRun	:= FALSE;
			bHermesStop	:= TRUE;
		END_IF

		IF bHermesRun = TRUE THEN
			p_eAct	:= HermesActBGStartRun;

			IF (eStat = HermesActBGStartRun) AND (eStatus = Done) THEN
				p_eAct		:= HermesActIdle;
				bHermesRun	:= FALSE;
			END_IF
		END_IF

		IF bHermesStop = TRUE THEN
			p_eAct	:= HermesActBGStopRun;

			IF (eStat = HermesActBGStopRun) AND (eStatus = Done) THEN
				p_eAct		:= HermesActIdle;
				bHermesStop	:= FALSE;
			END_IF
		END_IF

	END_IF

	//Delete Old Log Files for 24 hours After Machine is Continuous Running 30 Days.

	fbDlyTmr(IN := TRUE);
	IF fbDlyTmr.Q THEN
		fbDeleteLogTmr (IN := TRUE);
		IF fbDeleteLogTmr.Q AND eStatus <> Busy THEN
			p_eAct := HermesActDeleteOldLog;
			IF eStat = HermesActDeleteOldLog AND eStatus = Done THEN
				p_eAct := HermesActIdle;
				fbDlyTmr (IN := FALSE);
				fbDeleteLogTmr (IN := FALSE);
			END_IF
		END_IF
	END_IF
END_ACTION
```

#### Act_Link.st - Change By Project
```iecst
(** 2021-08-01 **)
ACTION Act_Link:

	//Receive Alive Time
	p_tyParam.tRcvAlive	:= p_tyParam.tSndAlive * 2;

	//Ready Send
	//Transfer Finished
//	IF (p_eLinkConvDir = ConvDirLToR) OR (p_eLinkConvDir = ConvDirRToR) THEN
		IF EDGENEG(p_bFirstZoneEndSen) THEN
			p_bSndCompl	:= TRUE;
		END_IF
//	ELSE
//		IF EDGENEG(p_bLinkDILeftSen) THEN
//			p_bSndCompl	:= TRUE;
//		END_IF
//	END_IF

	//Good Bad Board
//	IF p_bLinkOpsConvGdBrd = TRUE THEN
		p_eFailedBoard	:= HermesGoodBoard;
//	ELSE
//		p_eFailedBoard	:= HermesFailedBoard;
//	END_IF

	//New Product for Board Forecast(Id)
	//p_bNewProduct will be True only when machine accepted new recipe, can perform ChangeOver, i.e Machine Free (all zones).
//	p_bNewProduct := ((EDGEPOS(p_bLinkProdRcpCurrAll[0].sRcpNm = p_bLinkProdRcpCurrAll[1].sRcpNm)) AND (p_bLinkStartupRun = FALSE));

	//p_bNewWidth will be True only when machine accepted new width, can perform ChangeOver, i.e Machine Free (all zones).
//	p_bNewWidth := ((EDGEPOS(p_bLinkProdRcpCurrAll[0].diWidthInUM = p_bLinkProdRcpCurrAll[1].diWidthInUM)) AND (p_bLinkStartupRun = FALSE));

	p_bRdySnd	:= p_bLinkOpsTravLifLDDSComm AND p_eLinkTravLifLDPosGo = TravLifLDPosDS2;

	//Machine Cycle Time
	p_rMcCycleTm ACCESS p_NtParamDSHermesMcCycleTm; //Change this if machine got Worst/Least/Different Cycle Time accordingly

	//Flipped Board
	p_eFlippedBoard	:= USINT_TO_UDINT(p_usiLinkProdRcpCurrRcpFlipBrd);

	//Machine All Empty(for ChangeOver), adjust accordingly                                                            //Add
	bAllZonesEmpty := p_bOpsGConv1HvBrd = FALSE AND p_bFirstZoneEndSen = FALSE;// AND p_bLinkDIPresentSen = FALSE (*AND p_tyDI.bTopCoverSWSig = TRUE*);

	//Machine First Zone have board
	p_bFirstZoneHaveBoard := (p_bUSHermesStopTransport AND p_bOpsGConv1HvBrd) OR (p_bOpsGConv1HvBrd AND p_bUSHermesTransporting = FALSE); //Zone 1 have board, either PCB_In from upstream Or Manually load PCB at Zone 1

END_ACTION
```

#### Act_Background_ProcessData.st - Do Not Change!!!
```iecst
(** 2021-08-01 **)
ACTION Act_Background_ProcessData:

	//Pass Board Available data and TransportFinished BOOL to "BoardDeparted" (SupervisoryHermes)

	tyBoardDepartedInfo := tyBoardAvailableSnd;

	IF EDGEPOS (fbSequenceDS.eMsgTypeSnd = HermesMsgTypeTransportFinished) THEN
		bTransportFinishedSnd := TRUE;
	END_IF

	//Auto Reset bTransportFinishedSnd
	fbSendTm(IN := bTransportFinishedSnd, PT := T#0.3S);
	IF fbSendTm.Q = TRUE THEN
		fbSendTm(IN := FALSE);

		bTransportFinishedSnd	:= FALSE;
	END_IF

	//For Power On or Transfer New Program, udiBAIndex will reset to 0. To find which array sBoardId is empty and continue writing.
	IF udiBAIndex = 0 AND p_bLinkStartupRun = FALSE THEN

		udiTargetAddress := ADR(a_tyBoardDepartedInfo[0].tyData.sBoardId); //Start address
		udiSizeAddress   := SIZEOF(a_tyBoardDepartedInfo[0]); //Size of one array

		FOR i := 0 TO 49 DO //50 Boards Data

			IF memcmp((udiTargetAddress)+(i*udiSizeAddress), ADR('') , 1) = 0 THEN

				bFoundIndex	:= TRUE;
				udiBAIndex := i;
				EXIT;
			END_IF

		END_FOR
	END_IF

	//Retain last 50 PCB handled Boards Data
	p_udiRetainDataAddr	:= ADR(a_tyBoardDepartedInfo);
	p_udiRetainDataLen	:= SIZEOF(a_tyBoardDepartedInfo);

	//Write BoardAvailable Data into arrays and store after send out TransportFinished
	IF EDGENEG(bTransportFinishedSnd) THEN

		memset(ADR(a_tyBoardDepartedInfo[udiBAIndex]) , 0 , SIZEOF(a_tyBoardDepartedInfo[udiBAIndex]));
		memcpy(ADR(a_tyBoardDepartedInfo[udiBAIndex]) , ADR(tyBoardDepartedInfo) , SIZEOF(tyBoardDepartedInfo));

		udiBAIndex	:= udiBAIndex + 1;

		p_eAct := HermesActWriteRetain;

	END_IF

	IF eStatus = Done AND eStat = HermesActWriteRetain THEN
		p_eAct		:= HermesActIdle;
	END_IF

	IF udiBAIndex >= 50 THEN
	   udiBAIndex := 0;
	END_IF

	//BoardForecast
	bFeatureBoardForecast := (p_tyParam.bFeatureBoardForecast = TRUE) AND (tyServiceDescriptionRcv.tyAvl.tySupportedFeatures.bFeatureBoardForecast = TRUE) (*AND bHandshakeDone*) ;

	//New Product can come anytime from Upstream / Select From Product Setting
	IF EDGEPOS (p_bNewProduct) THEN //p_bNewProduct will be True only when machine accepted new recipe, can perform ChangeOver, i.e Machine Free (all zones).
		bNewChangeOver := TRUE;
		idxBoardForecastId	:= 0;//index to send B.F(Id)
	END_IF

	//New Width
	IF EDGEPOS (p_bNewWidth) THEN //p_bSiemensNewProduct will be True only when machine accepted new recipe, can perform ChangeOver, i.e Machine Free (all zones).
		bNewChangeOver := TRUE;
		idxBoardForecastId	:= 0;//index to send B.F(Id)
	END_IF

	IF bFeatureBoardForecast = TRUE THEN
		IF bNewChangeOver AND bAllZonesEmpty AND p_bInitDone THEN //Machine Free (all zones)
			bSendBFId := TRUE;
			bNewChangeOver := FALSE;
		END_IF
	ELSE
		bNewChangeOver := FALSE;
		bSendBFId := FALSE;
		bRstSendBFId := FALSE;
		idxBoardForecastId	    := 0;
		idxBoardForecastNoId	:= 0;
	END_IF

	//Reset bSendBFId and idxBoardForecastId	after receive Machine Ready(Id) or Machine Ready()
	IF bRstSendBFId THEN
		bSendBFId := FALSE;
		bRstSendBFId := FALSE;
		idxBoardForecastId	:= 0;
	END_IF

//	//Reset both idxBoardForecastId under handshake condition. Note: idxBoardForecastId only send once.
//	IF (fbSequenceDS.eState <> HermesStateNotAvailableNotReady) AND (fbSequenceDS.eState <> HermesStateMachineReady) AND (fbSequenceDS.eState <> HermesStateBoardAvailable) AND (fbSequenceDS.eState <> HermesStateAvailableAndReady) AND bHandshakeDone = TRUE THEN
//		idxBoardForecastId	:= 0;//index to send B.F(Id)
//	END_IF

	//Reset idxBoardForecastNoId when incoming zone empty
	IF p_bFirstZoneHaveBoard =FALSE AND p_bFirstZoneEndSen = FALSE THEN
		idxBoardForecastNoId	:= 0;//index to send B.F()
	END_IF

END_ACTION
```

#### Act_Background_CmpParamRcv.st - Do Not Change!!!
```iecst
(** 2021-08-01 **)
ACTION Act_Background_CmpParamRcv:

	IF eStatus2 <> Error THEN

		IF tyMsgTypeRcv.bStopTransport = TRUE THEN
			udiStatus2	:= fHermesChkParamSTST(tyStartTransport , tyStopTransport);

			IF udiStatus2 <> 0 THEN
				eStatus2	:= Error;

				IF udiStatus2 = 2712 THEN
					udiStatus2	:= 10104;	//BoardId Mismatch While Checking Start Transport & Stop Transport
				ELSIF udiStatus2 = 2713 THEN
					udiStatus2	:= 10105;	//BoardId Missing While Checking Start Transport & Stop Transport
				END_IF

				fHermesAddOneMsgSend(ADR(a_eMsgSend) , ADR(udiMsgSendBffr) , HermesMsgTypeNotification);

				tyNotificationSnd.tyAvl.bSeverity			:= TRUE;
				tyNotificationSnd.tyAvl.bNotificationCode	:= TRUE;
				tyNotificationSnd.tyAvl.bDescription		:= TRUE;
				tyNotificationSnd.tyData.eSeverity			:= HermesSeverityFatalError;
				tyNotificationSnd.tyData.iNotificationCode	:= UDINT_TO_INT(udiStatus2);
				tyNotificationSnd.tyData.sDescription		:= a_tyAlmText[udiStatus2].sAlmText;
			END_IF
		END_IF

		IF tyMsgTypeRcv.bStartTransport = TRUE THEN
			IF fHermesChkParamBAST(tyBoardAvailableSnd , tyStartTransport) <> 0 THEN
					p_bSndNotStart	:= TRUE;
			END_IF
		END_IF

	    IF bFeatureBoardForecast THEN
			IF tyMsgTypeRcv.bMachineReady = TRUE AND bSendBFId AND (idxBoardForecastId = 1) THEN
				udiStatus2	:= fHermesChkParamBFMR(tyBoardForecastSnd , tyMachineReady); //Modify this if our machine need to Error when ForecastId in MachineReady(Id) received is different

				IF udiStatus2 <> 0 THEN
					eStatus2	:= Error;

					IF udiStatus2 = 2716 THEN
						udiStatus2	:= 10164;	//Forecast Id Mismatch While Checking BoardForecast & Machine Ready
					ELSIF udiStatus2 = 2717 THEN
						udiStatus2	:= 10165;	//Product Type Id Mismatch While Checking BoardForecast & Machine Ready
					ELSIF udiStatus2 = 2718 THEN
						udiStatus2	:= 10166;	//Width Mismatch While Checking BoardForecast & Machine Ready
					END_IF

					fHermesAddOneMsgSend(ADR(a_eMsgSend) , ADR(udiMsgSendBffr) , HermesMsgTypeNotification);

					tyNotificationSnd.tyAvl.bSeverity			:= TRUE;
					tyNotificationSnd.tyAvl.bNotificationCode	:= TRUE;
					tyNotificationSnd.tyAvl.bDescription		:= TRUE;
					tyNotificationSnd.tyData.eSeverity			:= HermesSeverityFatalError; //Let it Fatal and reset connection
					tyNotificationSnd.tyData.iNotificationCode	:= UDINT_TO_INT(udiStatus2);
					tyNotificationSnd.tyData.sDescription		:= a_tyAlmText[udiStatus2].sAlmText;

				ELSE
					bRstSendBFId := TRUE; //Reset bSendBFId if MachineReady(Id) or MachineReady() received is ok
				END_IF
			END_IF
		END_IF
	END_IF

END_ACTION
```

#### Act_Background_Sequence.st - Do Not Change!!!
```iecst
 (** 2021-08-01 **)
ACTION Act_Background_Sequence:

	IF eStatus1 <> Error THEN

		IF p_bOpsRun = FALSE THEN
			p_bSndIncompl	:= TRUE;
		END_IF

		IF tyMsgTypeRcv.bStopTransport = TRUE THEN
			IF tyStopTransport.tyData.eTransferState = HermesTransferStateNotStarted THEN
				p_bSndNotStart	:= TRUE;
			ELSIF tyStopTransport.tyData.eTransferState = HermesTransferStateIncomplete THEN
				p_bSndIncompl	:= TRUE;
			END_IF
		END_IF

		//Sequence
		fbSequenceDS.bRstState		        := bRstState;
		fbSequenceDS.bRdySnd	        	:= p_bRdySnd; //Machine in OpsG step DSCommTmr (Have DBA)
		fbSequenceDS.bSndCompl	        	:= p_bSndCompl; //Send TransportFinished Msg = Complete (Value = 3)
		fbSequenceDS.bSndIncompl        	:= p_bSndIncompl; //Send TransportFinished Msg = Incomplete (Value = 2)
		fbSequenceDS.bSndNotStart        	:= p_bSndNotStart; //Send TransportFinished Msg = Not Started (Value = 1)
		fbSequenceDS.bFeatureBoardForecast	:= bFeatureBoardForecast; //Feature BoardForecast
		fbSequenceDS.bOpsRun	        	:= p_bOpsRun; //Machine in AutoMode
		fbSequenceDS.bSendBFId              := bSendBFId; //Send B.F with forecast ID, then block Hermes.eState until Downstream reply a MachineReady(Id) or MachineReady()
		fbSequenceDS.bFirstZoneHaveBoard	:= p_bFirstZoneHaveBoard; //First Zone Have Board
		fbSequenceDS.bFirstZoneEndSen	    := p_bFirstZoneEndSen; //First Zone End sensor
		fbSequenceDS.bAllZonesEmpty	        := bAllZonesEmpty; //All Zones empty
		fbSequenceDS(bEn := TRUE);
		bUSRdy		                       	:= fbSequenceDS.bUSRdy;
		bDSRdy			                    := fbSequenceDS.bDSRdy;
		bTransporting                      	:= fbSequenceDS.bTransporting;
		bStopTransport                     	:= fbSequenceDS.bStopTransport;

		IF EDGEPOS(tyMsgTypeRcv.bMachineReady = TRUE) THEN
			bRstSendBFId := TRUE;
		END_IF

		bUSGdRdy	:= (tyBoardAvailableSnd.tyAvl.bFailedBoard = FALSE) OR ((tyBoardAvailableSnd.tyAvl.bFailedBoard = TRUE) AND (tyBoardAvailableSnd.tyData.eFailedBoard <> HermesFailedBoard));

		bDSGdRdy	:= (tyMachineReady.tyAvl.bFailedBoard = FALSE) OR ((tyMachineReady.tyAvl.bFailedBoard = TRUE) AND (tyMachineReady.tyData.eFailedBoard <> HermesFailedBoard));

		IF fbSequenceDS.eState >= HermesStateNotAvailableNotReady THEN
			bHandshakeDone	:= TRUE;
		ELSE
			bHandshakeDone	:= FALSE;
		END_IF

		IF EDGEPOS(fbSequenceDS.eState = HermesStateTransporting) THEN
			p_bSndCompl		:= FALSE;
			p_bSndIncompl	:= FALSE;
			p_bSndNotStart	:= FALSE;
		END_IF

		IF fbSequenceDS.eMsgTypeSnd = HermesMsgTypeServiceDescription THEN
			fHermesAddOneMsgSend(ADR(a_eMsgSend) , ADR(udiMsgSendBffr) , HermesMsgTypeServiceDescription);

			tyServiceDescriptionSnd.tyData.sMachineId								    	:= p_sMcId;
			tyServiceDescriptionSnd.tyData.iLaneId											:= p_tyParam.iLaneID;
			tyServiceDescriptionSnd.tyData.sInterfaceId										:= p_tyParam.sDownstreamInterfaceId;
			tyServiceDescriptionSnd.tyData.sVersion											:= p_sVersion;
			tyServiceDescriptionSnd.tyData.tySupportedFeatures.bFeatureCheckAliveResponse	:= (p_tyParam.bFeatureCheckAliveResponse) AND (p_tyParam.tRcvAlive <> T#0s) AND (p_tyParam.tSndAlive <> T#0s);
			tyServiceDescriptionSnd.tyData.tySupportedFeatures.bFeatureBoardForecast		:= p_tyParam.bFeatureBoardForecast;
			tyServiceDescriptionSnd.tyData.tySupportedFeatures.bFeatureQueryBoardInfo		:= FALSE;
			tyServiceDescriptionSnd.tyData.tySupportedFeatures.bFeatureSendBoardInfo		:= p_tyParam.bFeatureSendBoardInfo;
			tyServiceDescriptionSnd.tyAvl.bMachineId										:= tyServiceDescriptionSnd.tyData.sMachineId <> '';
			tyServiceDescriptionSnd.tyAvl.bLaneId											:= tyServiceDescriptionSnd.tyData.iLaneId<>0;
			tyServiceDescriptionSnd.tyAvl.bInterfaceId										:= tyServiceDescriptionSnd.tyData.sInterfaceId <> '';
			tyServiceDescriptionSnd.tyAvl.bVersion											:= TRUE;
			tyServiceDescriptionSnd.tyAvl.bSupportedFeatures								:= p_tyParam.bFeatureCheckAliveResponse OR p_tyParam.bFeatureBoardForecast OR p_tyParam.bFeatureSendBoardInfo;
			tyServiceDescriptionSnd.tyAvl.tySupportedFeatures.bFeatureCheckAliveResponse	:= (p_tyParam.bFeatureCheckAliveResponse) AND (p_tyParam.tRcvAlive <> T#0s) AND (p_tyParam.tSndAlive <> T#0s);
			tyServiceDescriptionSnd.tyAvl.tySupportedFeatures.bFeatureBoardForecast			:= p_tyParam.bFeatureBoardForecast;
			tyServiceDescriptionSnd.tyAvl.tySupportedFeatures.bFeatureQueryBoardInfo		:= FALSE;
			tyServiceDescriptionSnd.tyAvl.tySupportedFeatures.bFeatureSendBoardInfo			:= p_tyParam.bFeatureSendBoardInfo;

		ELSIF fbSequenceDS.eMsgTypeSnd = HermesMsgTypeBoardForecastId THEN //Beside of sProductTypeId, rWidth, other parameters use default. If upstream does not support BoardForecast, then our machine has no data.

			IF p_eLinkCustomerReq = Siemens AND p_sWorkOrderId <> '' AND  (p_usiProdRcpCurrRcp1McMod = 1) THEN

				IF (idxBoardForecastId < 1) THEN

					fHermesAddOneMsgSend(ADR(a_eMsgSend) , ADR(udiMsgSendBffr) , HermesMsgTypeBoardForecast);
					fHermesGenerateUUID(ADR(tyBoardForecastSnd.tyData.sForecastId) , p_tyDTStructure , pa_usiMacAddr); //Generate ForecastID if there is new Product Changeover

					idxBoardForecastId := idxBoardForecastId + 1;

				END_IF

				tyBoardForecastSnd.tyData.rTimeUntilAvailable       := p_rMcCycleTm + p_rAWCycleTm;
				tyBoardForecastSnd.tyData.sBoardId 			        := ''; //no need to send BoardId for HermesMsgTypeBoardForecastId.
				tyBoardForecastSnd.tyData.sBoardIdCreatedBy			:= ''; //no need to send BoardIdCreatedBy since no BoardId.
				tyBoardForecastSnd.tyData.eFailedBoard				:= p_eFailedBoard;
				tyBoardForecastSnd.tyData.sProductTypeId			:= p_tySendWorkOrderData.tyData.sProductTypeId;
				tyBoardForecastSnd.tyData.eFlippedBoard		    	:= p_eFlippedBoard;
				tyBoardForecastSnd.tyData.sTopBarcode				:= p_sTopBarcode;
				tyBoardForecastSnd.tyData.sBottomBarcode			:= p_sBottomBarcode;
				tyBoardForecastSnd.tyData.rLength					:= p_tySendWorkOrderData.tyData.rLength;
				tyBoardForecastSnd.tyData.rWidth					:= p_tySendWorkOrderData.tyData.rWidth;
				tyBoardForecastSnd.tyData.rThickness				:= p_tySendWorkOrderData.tyData.rThickness;
				tyBoardForecastSnd.tyData.rConveyorSpeed			:= p_rConveyorSpeed; //dont have
				tyBoardForecastSnd.tyData.rTopClearanceHeight		:= p_tySendWorkOrderData.tyData.rTopClearanceHeight;
				tyBoardForecastSnd.tyData.rBottomClearanceHeight	:= p_tySendWorkOrderData.tyData.rBottomClearanceHeight;
				tyBoardForecastSnd.tyData.rWeight					:= p_tySendWorkOrderData.tyData.rWeight;
				tyBoardForecastSnd.tyData.sWorkOrderId			    := p_tySendWorkOrderData.tyData.sWorkOrderId;
				tyBoardForecastSnd.tyData.sBatchId		            := p_tySendWorkOrderData.tyData.sBatchId;

				tyBoardForecastSnd.tyAvl.bForecastId 			    := TRUE;
				tyBoardForecastSnd.tyAvl.bTimeUntilAvailable		:= tyBoardForecastSnd.tyData.rTimeUntilAvailable <> 0;
				tyBoardForecastSnd.tyAvl.bBoardId 				    := tyBoardForecastSnd.tyData.sBoardId <> '';
				tyBoardForecastSnd.tyAvl.bBoardIdCreatedBy 		    := TRUE;
				tyBoardForecastSnd.tyAvl.bFailedBoard 			    := TRUE;
				tyBoardForecastSnd.tyAvl.bProductTypeId 			:= tyBoardForecastSnd.tyData.sProductTypeId <> '';
				tyBoardForecastSnd.tyAvl.bFlippedBoard 			    := TRUE;
				tyBoardForecastSnd.tyAvl.bTopBarcode 			    := tyBoardForecastSnd.tyData.sTopBarcode <> '';
				tyBoardForecastSnd.tyAvl.bBottomBarcode 			:= tyBoardForecastSnd.tyData.sBottomBarcode <> '';
				tyBoardForecastSnd.tyAvl.bLength 				    := tyBoardForecastSnd.tyData.rLength <> 0;
				tyBoardForecastSnd.tyAvl.bWidth 				    := tyBoardForecastSnd.tyData.rWidth <> 0 AND (p_bBFWidthEn = TRUE);
				tyBoardForecastSnd.tyAvl.bThickness 			    := tyBoardForecastSnd.tyData.rThickness <> 0 AND (p_bBFSltEn = TRUE);
				tyBoardForecastSnd.tyAvl.bConveyorSpeed 			:= tyBoardForecastSnd.tyData.rConveyorSpeed <> 0;
				tyBoardForecastSnd.tyAvl.bTopClearanceHeight 		:= tyBoardForecastSnd.tyData.rTopClearanceHeight <> 0 AND (p_bBFSltEn = TRUE);
				tyBoardForecastSnd.tyAvl.bBottomClearanceHeight 	:= tyBoardForecastSnd.tyData.rBottomClearanceHeight <> 0 AND (p_bBFSltEn = TRUE);
				tyBoardForecastSnd.tyAvl.bWeight 			    	:= tyBoardForecastSnd.tyData.rWeight <> 0;
				tyBoardForecastSnd.tyAvl.bWorkOrderId 		    	:= tyBoardForecastSnd.tyData.sWorkOrderId <> '';
				tyBoardForecastSnd.tyAvl.bBatchId 		        	:= tyBoardForecastSnd.tyData.sBatchId <> '';
			ELSE
				IF (idxBoardForecastId < 1) THEN

					fHermesAddOneMsgSend(ADR(a_eMsgSend) , ADR(udiMsgSendBffr) , HermesMsgTypeBoardForecast);
					fHermesGenerateUUID(ADR(tyBoardForecastSnd.tyData.sForecastId) , p_tyDTStructure , pa_usiMacAddr); //Generate ForecastID if there is new Product Changeover

					idxBoardForecastId := idxBoardForecastId + 1;

				END_IF

				tyBoardForecastSnd.tyData.rTimeUntilAvailable       := p_rMcCycleTm + p_rAWCycleTm;
				tyBoardForecastSnd.tyData.sBoardId 			        := ''; //no need to send BoardId for HermesMsgTypeBoardForecastId.
				tyBoardForecastSnd.tyData.sBoardIdCreatedBy			:= ''; //no need to send BoardIdCreatedBy since no BoardId.
				tyBoardForecastSnd.tyData.eFailedBoard 			    := p_eFailedBoard;
				tyBoardForecastSnd.tyData.sProductTypeId 			:= p_sRecipeNm; //recipe0 name = running recipe name
				tyBoardForecastSnd.tyData.eFlippedBoard 			:= p_eFlippedBoard;
				tyBoardForecastSnd.tyData.sTopBarcode 		    	:= p_sTopBarcode;
				tyBoardForecastSnd.tyData.sBottomBarcode 			:= p_sBottomBarcode;
				tyBoardForecastSnd.tyData.rLength 				    := p_rLength;
				tyBoardForecastSnd.tyData.rWidth 			    	:= DINT_TO_REAL(p_diWidthInUM) / 1000; //recipe 0 width	 = running recipe width
				tyBoardForecastSnd.tyData.rThickness 		    	:= p_rThickness;
				tyBoardForecastSnd.tyData.rConveyorSpeed 			:= p_rConveyorSpeed;
				tyBoardForecastSnd.tyData.rTopClearanceHeight 		:= p_rTopClearanceHeight;
				tyBoardForecastSnd.tyData.rBottomClearanceHeight 	:= p_rBottomClearanceHeight;
				tyBoardForecastSnd.tyData.rWeight 			    	:= p_rWeight;
//				tyBoardForecastSnd.tyData.sWorkOrderId 			    := p_sWorkOrderId;
//				tyBoardForecastSnd.tyData.sBatchId 			        := p_sBatchId;
				tyBoardForecastSnd.tyData.sWorkOrderId 			    := '';
				tyBoardForecastSnd.tyData.sBatchId 			        := '';

				tyBoardForecastSnd.tyAvl.bForecastId 			    := TRUE;
				tyBoardForecastSnd.tyAvl.bTimeUntilAvailable		:= tyBoardForecastSnd.tyData.rTimeUntilAvailable <> 0;
				tyBoardForecastSnd.tyAvl.bBoardId 				    := tyBoardForecastSnd.tyData.sBoardId <> '';
				tyBoardForecastSnd.tyAvl.bBoardIdCreatedBy 		    := TRUE;
				tyBoardForecastSnd.tyAvl.bFailedBoard 			    := TRUE;
				tyBoardForecastSnd.tyAvl.bProductTypeId 			:= tyBoardForecastSnd.tyData.sProductTypeId <> '';
				tyBoardForecastSnd.tyAvl.bFlippedBoard 			    := TRUE;
				tyBoardForecastSnd.tyAvl.bTopBarcode 			    := tyBoardForecastSnd.tyData.sTopBarcode <> '';
				tyBoardForecastSnd.tyAvl.bBottomBarcode 			:= tyBoardForecastSnd.tyData.sBottomBarcode <> '';
				tyBoardForecastSnd.tyAvl.bLength 				    := tyBoardForecastSnd.tyData.rLength <> 0;
				tyBoardForecastSnd.tyAvl.bWidth 				    := tyBoardForecastSnd.tyData.rWidth <> 0 AND (p_bBFWidthEn = TRUE);
				tyBoardForecastSnd.tyAvl.bThickness 			    := tyBoardForecastSnd.tyData.rThickness <> 0 AND (p_bBFSltEn = TRUE);
				tyBoardForecastSnd.tyAvl.bConveyorSpeed 			:= tyBoardForecastSnd.tyData.rConveyorSpeed <> 0;
				tyBoardForecastSnd.tyAvl.bTopClearanceHeight 		:= tyBoardForecastSnd.tyData.rTopClearanceHeight <> 0 AND (p_bBFSltEn = TRUE);
				tyBoardForecastSnd.tyAvl.bBottomClearanceHeight 	:= tyBoardForecastSnd.tyData.rBottomClearanceHeight <> 0 AND (p_bBFSltEn = TRUE);
				tyBoardForecastSnd.tyAvl.bWeight 			    	:= tyBoardForecastSnd.tyData.rWeight <> 0;
				tyBoardForecastSnd.tyAvl.bWorkOrderId 		    	:= tyBoardForecastSnd.tyData.sWorkOrderId <> '';
				tyBoardForecastSnd.tyAvl.bBatchId 		        	:= tyBoardForecastSnd.tyData.sBatchId <> '';
			END_IF

		ELSIF fbSequenceDS.eMsgTypeSnd = HermesMsgTypeBoardForecastNoId THEN

			IF p_eLinkCustomerReq = Siemens AND p_sWorkOrderId <> '' AND (p_usiProdRcpCurrRcp1McMod = 1)  THEN

				IF p_bNewBrdAvlFirstZone THEN //Generate BoardForecast() by our machine for Manual Load Board at First Zone

					IF (idxBoardForecastNoId < 1) THEN

						fHermesAddOneMsgSend(ADR(a_eMsgSend) , ADR(udiMsgSendBffr) , HermesMsgTypeBoardForecast);

						idxBoardForecastNoId := idxBoardForecastNoId + 1;

					END_IF

					tyBoardForecastSnd.tyData.sForecastId		        := ''; //Do not need to generate ForecastID to downstream

					IF idxBoardForecastNoId <= 1 THEN
						tyBoardForecastSnd.tyData.rTimeUntilAvailable	:= p_rMcCycleTm;
						//				ELSIF idxBoardForecastNoId = 2 THEN
						//					tyBoardForecastSnd.tyData.rTimeUntilAvailable	:= p_rMcCycleTm - (p_rMcCycleTm/3); //divide B.F to 3 segments, open up if needed
						//				ELSIF idxBoardForecastNoId = 3 THEN
						//					tyBoardForecastSnd.tyData.rTimeUntilAvailable	:= p_rMcCycleTm - ((p_rMcCycleTm/3)*2);
					END_IF

					fHermesGenerateUUID(ADR(tyBoardForecastSnd.tyData.sBoardId) , p_tyDTStructure , pa_usiMacAddr);

                    tyBoardForecastSnd.tyData.sBoardIdCreatedBy			:= p_sMcId; //no need to send BoardIdCreatedBy since no BoardId.
					tyBoardForecastSnd.tyData.eFailedBoard				:= p_eFailedBoard;
					tyBoardForecastSnd.tyData.sProductTypeId			:= p_tySendWorkOrderData.tyData.sProductTypeId;
					tyBoardForecastSnd.tyData.eFlippedBoard		    	:= p_eFlippedBoard;
					tyBoardForecastSnd.tyData.sTopBarcode				:= p_sTopBarcode;
					tyBoardForecastSnd.tyData.sBottomBarcode			:= p_sBottomBarcode;
					tyBoardForecastSnd.tyData.rLength					:= p_tySendWorkOrderData.tyData.rLength;
					tyBoardForecastSnd.tyData.rWidth					:= p_tySendWorkOrderData.tyData.rWidth;
					tyBoardForecastSnd.tyData.rThickness				:= p_tySendWorkOrderData.tyData.rThickness;
					tyBoardForecastSnd.tyData.rConveyorSpeed			:= p_rConveyorSpeed; //dont have
					tyBoardForecastSnd.tyData.rTopClearanceHeight		:= p_tySendWorkOrderData.tyData.rTopClearanceHeight;
					tyBoardForecastSnd.tyData.rBottomClearanceHeight	:= p_tySendWorkOrderData.tyData.rBottomClearanceHeight;
					tyBoardForecastSnd.tyData.rWeight					:= p_tySendWorkOrderData.tyData.rWeight;
					tyBoardForecastSnd.tyData.sWorkOrderId			    := p_tySendWorkOrderData.tyData.sWorkOrderId;
					tyBoardForecastSnd.tyData.sBatchId		            := p_tySendWorkOrderData.tyData.sBatchId;

					tyBoardForecastSnd.tyAvl.bForecastId 			    := tyBoardForecastSnd.tyData.sForecastId <> '';
					tyBoardForecastSnd.tyAvl.bTimeUntilAvailable		:= tyBoardForecastSnd.tyData.rTimeUntilAvailable <> 0;
					tyBoardForecastSnd.tyAvl.bBoardId 				    := tyBoardForecastSnd.tyData.sBoardId <> '';
					tyBoardForecastSnd.tyAvl.bBoardIdCreatedBy 	    	:= tyBoardForecastSnd.tyData.sBoardIdCreatedBy <> '';
					tyBoardForecastSnd.tyAvl.bFailedBoard 			    := TRUE;
					tyBoardForecastSnd.tyAvl.bProductTypeId 			:= tyBoardForecastSnd.tyData.sProductTypeId <> '';
					tyBoardForecastSnd.tyAvl.bFlippedBoard 		    	:= TRUE;
					tyBoardForecastSnd.tyAvl.bTopBarcode 			    := tyBoardForecastSnd.tyData.sTopBarcode <> '';
					tyBoardForecastSnd.tyAvl.bBottomBarcode 			:= tyBoardForecastSnd.tyData.sBottomBarcode <> '';
					tyBoardForecastSnd.tyAvl.bLength 				    := tyBoardForecastSnd.tyData.rLength <> 0;
					tyBoardForecastSnd.tyAvl.bWidth 				    := tyBoardForecastSnd.tyData.rWidth <> 0 AND (p_bBFWidthEn = TRUE);
					tyBoardForecastSnd.tyAvl.bThickness 			    := tyBoardForecastSnd.tyData.rThickness <> 0 AND (p_bBFSltEn = TRUE);
					tyBoardForecastSnd.tyAvl.bConveyorSpeed 			:= tyBoardForecastSnd.tyData.rConveyorSpeed <> 0;
					tyBoardForecastSnd.tyAvl.bTopClearanceHeight 		:= tyBoardForecastSnd.tyData.rTopClearanceHeight <>0 AND (p_bBFSltEn = TRUE);
					tyBoardForecastSnd.tyAvl.bBottomClearanceHeight 	:= tyBoardForecastSnd.tyData.rBottomClearanceHeight <>0 AND (p_bBFSltEn = TRUE);
					tyBoardForecastSnd.tyAvl.bWeight 			    	:= tyBoardForecastSnd.tyData.rWeight <> 0;
					tyBoardForecastSnd.tyAvl.bWorkOrderId 		    	:= tyBoardForecastSnd.tyData.sWorkOrderId <> '';
					tyBoardForecastSnd.tyAvl.bBatchId 		        	:= tyBoardForecastSnd.tyData.sBatchId <> '';

				ELSE //take PCB_In Board data (For PCB Transfer in from upstream)

					IF (idxBoardForecastNoId < 1) THEN

						fHermesAddOneMsgSend(ADR(a_eMsgSend) , ADR(udiMsgSendBffr) , HermesMsgTypeBoardForecast);
						idxBoardForecastNoId := idxBoardForecastNoId + 1;

					END_IF

					tyBoardForecastSnd.tyData.sForecastId		            := ''; //Do not need to generate ForecastID to downstream

					IF idxBoardForecastNoId <= 1 THEN
						tyBoardForecastSnd.tyData.rTimeUntilAvailable	    := p_rMcCycleTm;
						//			    ELSIF idxBoardForecastNoId = 2 THEN
						//					tyBoardForecastSnd.tyData.rTimeUntilAvailable    	:= p_rMcCycleTm - (p_rMcCycleTm/3); //divide B.F to 3 segments, open up if needed
						//				ELSIF idxBoardForecastNoId = 3 THEN
						//					tyBoardForecastSnd.tyData.rTimeUntilAvailable	    := p_rMcCycleTm - ((p_rMcCycleTm/3)*2);
					END_IF

					tyBoardForecastSnd.tyData.sBoardId                  := p_tyUSBoardArrivedData.tyData.sBoardId;
					tyBoardForecastSnd.tyData.sBoardIdCreatedBy         := p_tyUSBoardArrivedData.tyData.sBoardIdCreatedBy;
					tyBoardForecastSnd.tyData.eFailedBoard 		    	:= p_tyUSBoardArrivedData.tyData.eFailedBoard;
					tyBoardForecastSnd.tyData.sProductTypeId 			:= p_tyUSBoardArrivedData.tyData.sProductTypeId;
					tyBoardForecastSnd.tyData.eFlippedBoard 			:= p_tyUSBoardArrivedData.tyData.eFlippedBoard;
					tyBoardForecastSnd.tyData.sTopBarcode 		    	:= p_tyUSBoardArrivedData.tyData.sTopBarcode;
					tyBoardForecastSnd.tyData.sBottomBarcode 			:= p_tyUSBoardArrivedData.tyData.sBottomBarcode;
					tyBoardForecastSnd.tyData.rLength 				    := p_tyUSBoardArrivedData.tyData.rLength;
					tyBoardForecastSnd.tyData.rWidth 			    	:= p_tyUSBoardArrivedData.tyData.rWidth;
					tyBoardForecastSnd.tyData.rThickness 		    	:= p_tyUSBoardArrivedData.tyData.rThickness;
					tyBoardForecastSnd.tyData.rConveyorSpeed 			:= p_tyUSBoardArrivedData.tyData.rConveyorSpeed;
					tyBoardForecastSnd.tyData.rTopClearanceHeight 		:= p_tyUSBoardArrivedData.tyData.rTopClearanceHeight;
					tyBoardForecastSnd.tyData.rBottomClearanceHeight 	:= p_tyUSBoardArrivedData.tyData.rBottomClearanceHeight;
					tyBoardForecastSnd.tyData.rWeight 			    	:= p_tyUSBoardArrivedData.tyData.rWeight;
					tyBoardForecastSnd.tyData.sWorkOrderId 		    	:= p_tyUSBoardArrivedData.tyData.sWorkOrderId;
					tyBoardForecastSnd.tyData.sBatchId 		        	:= p_tyUSBoardArrivedData.tyData.sBatchId;

					tyBoardForecastSnd.tyAvl.bForecastId 			    := tyBoardForecastSnd.tyData.sForecastId <> '';
					tyBoardForecastSnd.tyAvl.bTimeUntilAvailable		:= tyBoardForecastSnd.tyData.rTimeUntilAvailable <> 0;
					tyBoardForecastSnd.tyAvl.bBoardId 				    := tyBoardForecastSnd.tyData.sBoardId <> '';
					tyBoardForecastSnd.tyAvl.bBoardIdCreatedBy 	    	:= tyBoardForecastSnd.tyData.sBoardIdCreatedBy <> '';
					tyBoardForecastSnd.tyAvl.bFailedBoard 			    := TRUE;
					tyBoardForecastSnd.tyAvl.bProductTypeId 			:= tyBoardForecastSnd.tyData.sProductTypeId <> '';
					tyBoardForecastSnd.tyAvl.bFlippedBoard 		    	:= TRUE;
					tyBoardForecastSnd.tyAvl.bTopBarcode 			    := tyBoardForecastSnd.tyData.sTopBarcode <> '';
					tyBoardForecastSnd.tyAvl.bBottomBarcode 			:= tyBoardForecastSnd.tyData.sBottomBarcode <> '';
					tyBoardForecastSnd.tyAvl.bLength 				    := tyBoardForecastSnd.tyData.rLength <> 0;
					tyBoardForecastSnd.tyAvl.bWidth 				    := tyBoardForecastSnd.tyData.rWidth <> 0;
					tyBoardForecastSnd.tyAvl.bThickness 			    := tyBoardForecastSnd.tyData.rThickness <> 0;
					tyBoardForecastSnd.tyAvl.bConveyorSpeed 			:= tyBoardForecastSnd.tyData.rConveyorSpeed <> 0;
					tyBoardForecastSnd.tyAvl.bTopClearanceHeight 		:= tyBoardForecastSnd.tyData.rTopClearanceHeight <> 0;
					tyBoardForecastSnd.tyAvl.bBottomClearanceHeight 	:= tyBoardForecastSnd.tyData.rBottomClearanceHeight <> 0;
					tyBoardForecastSnd.tyAvl.bWeight 			    	:= tyBoardForecastSnd.tyData.rWeight <> 0;
					tyBoardForecastSnd.tyAvl.bWorkOrderId 		    	:= tyBoardForecastSnd.tyData.sWorkOrderId <> '';
					tyBoardForecastSnd.tyAvl.bBatchId 		        	:= tyBoardForecastSnd.tyData.sBatchId <> '';

				END_IF
			ELSE //no siemens

				IF p_bNewBrdAvlFirstZone THEN //Generate BoardForecast() by our machine for Manual Load Board at First Zone

					IF (idxBoardForecastNoId < 1) THEN

						fHermesAddOneMsgSend(ADR(a_eMsgSend) , ADR(udiMsgSendBffr) , HermesMsgTypeBoardForecast);

						idxBoardForecastNoId := idxBoardForecastNoId + 1;

					END_IF

					tyBoardForecastSnd.tyData.sForecastId		        := ''; //Do not need to generate ForecastID to downstream

					IF idxBoardForecastNoId <= 1 THEN
						tyBoardForecastSnd.tyData.rTimeUntilAvailable	:= p_rMcCycleTm;
						//				ELSIF idxBoardForecastNoId = 2 THEN
						//					tyBoardForecastSnd.tyData.rTimeUntilAvailable	:= p_rMcCycleTm - (p_rMcCycleTm/3); //divide B.F to 3 segments, open up if needed
						//				ELSIF idxBoardForecastNoId = 3 THEN
						//					tyBoardForecastSnd.tyData.rTimeUntilAvailable	:= p_rMcCycleTm - ((p_rMcCycleTm/3)*2);
					END_IF

					fHermesGenerateUUID(ADR(tyBoardForecastSnd.tyData.sBoardId) , p_tyDTStructure , pa_usiMacAddr);
					tyBoardForecastSnd.tyData.sBoardIdCreatedBy         := p_sMcId;
					tyBoardForecastSnd.tyData.eFailedBoard 		    	:= p_eFailedBoard;
					tyBoardForecastSnd.tyData.sProductTypeId 			:= p_sRecipeNm;	 //recipe 0 name = running recipe name
					tyBoardForecastSnd.tyData.eFlippedBoard 			:= p_eFlippedBoard;
					tyBoardForecastSnd.tyData.sTopBarcode 		    	:= p_sTopBarcode;
					tyBoardForecastSnd.tyData.sBottomBarcode 			:= p_sBottomBarcode;
					tyBoardForecastSnd.tyData.rLength 				    := p_rLength;
					tyBoardForecastSnd.tyData.rWidth 			    	:= DINT_TO_REAL(p_diWidthInUM) / 1000;	//recipe 0 width = running recipe width
					tyBoardForecastSnd.tyData.rThickness 		    	:= p_rThickness;
					tyBoardForecastSnd.tyData.rConveyorSpeed 			:= p_rConveyorSpeed;
					tyBoardForecastSnd.tyData.rTopClearanceHeight 		:= p_rTopClearanceHeight;
					tyBoardForecastSnd.tyData.rBottomClearanceHeight 	:= p_rBottomClearanceHeight;
					tyBoardForecastSnd.tyData.rWeight 			    	:= p_rWeight;
//					tyBoardForecastSnd.tyData.sWorkOrderId 		    	:= p_sWorkOrderId;
//					tyBoardForecastSnd.tyData.sBatchId	    	    	:= p_sBatchId;
					tyBoardForecastSnd.tyData.sWorkOrderId 		    	:= '';
					tyBoardForecastSnd.tyData.sBatchId	    	    	:= '';

					tyBoardForecastSnd.tyAvl.bForecastId 			    := tyBoardForecastSnd.tyData.sForecastId <> '';
					tyBoardForecastSnd.tyAvl.bTimeUntilAvailable		:= tyBoardForecastSnd.tyData.rTimeUntilAvailable <> 0;
					tyBoardForecastSnd.tyAvl.bBoardId 				    := tyBoardForecastSnd.tyData.sBoardId <> '';
					tyBoardForecastSnd.tyAvl.bBoardIdCreatedBy 	    	:= tyBoardForecastSnd.tyData.sBoardIdCreatedBy <> '';
					tyBoardForecastSnd.tyAvl.bFailedBoard 			    := TRUE;
					tyBoardForecastSnd.tyAvl.bProductTypeId 			:= tyBoardForecastSnd.tyData.sProductTypeId <> '';
					tyBoardForecastSnd.tyAvl.bFlippedBoard 		    	:= TRUE;
					tyBoardForecastSnd.tyAvl.bTopBarcode 			    := tyBoardForecastSnd.tyData.sTopBarcode <> '';
					tyBoardForecastSnd.tyAvl.bBottomBarcode 			:= tyBoardForecastSnd.tyData.sBottomBarcode <> '';
					tyBoardForecastSnd.tyAvl.bLength 				    := tyBoardForecastSnd.tyData.rLength <> 0;
					tyBoardForecastSnd.tyAvl.bWidth 				    := tyBoardForecastSnd.tyData.rWidth <> 0 AND (p_bBFWidthEn = TRUE);
					tyBoardForecastSnd.tyAvl.bThickness 			    := tyBoardForecastSnd.tyData.rThickness <> 0 AND (p_bBFSltEn = TRUE);
					tyBoardForecastSnd.tyAvl.bConveyorSpeed 			:= tyBoardForecastSnd.tyData.rConveyorSpeed <> 0;
					tyBoardForecastSnd.tyAvl.bTopClearanceHeight 		:= tyBoardForecastSnd.tyData.rTopClearanceHeight <>0 AND (p_bBFSltEn = TRUE);
					tyBoardForecastSnd.tyAvl.bBottomClearanceHeight 	:= tyBoardForecastSnd.tyData.rBottomClearanceHeight <>0 AND (p_bBFSltEn = TRUE);
					tyBoardForecastSnd.tyAvl.bWeight 			    	:= tyBoardForecastSnd.tyData.rWeight <> 0;
					tyBoardForecastSnd.tyAvl.bWorkOrderId 		    	:= tyBoardForecastSnd.tyData.sWorkOrderId <> '';
					tyBoardForecastSnd.tyAvl.bBatchId 		        	:= tyBoardForecastSnd.tyData.sBatchId <> '';

				ELSE //take PCB_In Board data (For PCB Transfer in from upstream)

					IF (idxBoardForecastNoId < 1) THEN

						fHermesAddOneMsgSend(ADR(a_eMsgSend) , ADR(udiMsgSendBffr) , HermesMsgTypeBoardForecast);
						idxBoardForecastNoId := idxBoardForecastNoId + 1;

					END_IF

					tyBoardForecastSnd.tyData.sForecastId		            := ''; //Do not need to generate ForecastID to downstream

					IF idxBoardForecastNoId <= 1 THEN
						tyBoardForecastSnd.tyData.rTimeUntilAvailable	    := p_rMcCycleTm;
						//			    ELSIF idxBoardForecastNoId = 2 THEN
						//					tyBoardForecastSnd.tyData.rTimeUntilAvailable    	:= p_rMcCycleTm - (p_rMcCycleTm/3); //divide B.F to 3 segments, open up if needed
						//				ELSIF idxBoardForecastNoId = 3 THEN
						//					tyBoardForecastSnd.tyData.rTimeUntilAvailable	    := p_rMcCycleTm - ((p_rMcCycleTm/3)*2);
					END_IF

					tyBoardForecastSnd.tyData.sBoardId                  := p_tyUSBoardArrivedData.tyData.sBoardId;
					tyBoardForecastSnd.tyData.sBoardIdCreatedBy         := p_tyUSBoardArrivedData.tyData.sBoardIdCreatedBy;
					tyBoardForecastSnd.tyData.eFailedBoard 		    	:= p_tyUSBoardArrivedData.tyData.eFailedBoard;
					tyBoardForecastSnd.tyData.sProductTypeId 			:= p_tyUSBoardArrivedData.tyData.sProductTypeId;
					tyBoardForecastSnd.tyData.eFlippedBoard 			:= p_tyUSBoardArrivedData.tyData.eFlippedBoard;
					tyBoardForecastSnd.tyData.sTopBarcode 		    	:= p_tyUSBoardArrivedData.tyData.sTopBarcode;
					tyBoardForecastSnd.tyData.sBottomBarcode 			:= p_tyUSBoardArrivedData.tyData.sBottomBarcode;
					tyBoardForecastSnd.tyData.rLength 				    := p_tyUSBoardArrivedData.tyData.rLength;
					tyBoardForecastSnd.tyData.rWidth 			    	:= p_tyUSBoardArrivedData.tyData.rWidth;
					tyBoardForecastSnd.tyData.rThickness 		    	:= p_tyUSBoardArrivedData.tyData.rThickness;
					tyBoardForecastSnd.tyData.rConveyorSpeed 			:= p_tyUSBoardArrivedData.tyData.rConveyorSpeed;
					tyBoardForecastSnd.tyData.rTopClearanceHeight 		:= p_tyUSBoardArrivedData.tyData.rTopClearanceHeight;
					tyBoardForecastSnd.tyData.rBottomClearanceHeight 	:= p_tyUSBoardArrivedData.tyData.rBottomClearanceHeight;
					tyBoardForecastSnd.tyData.rWeight 			    	:= p_tyUSBoardArrivedData.tyData.rWeight;
					tyBoardForecastSnd.tyData.sWorkOrderId 		    	:= p_tyUSBoardArrivedData.tyData.sWorkOrderId;
					tyBoardForecastSnd.tyData.sBatchId 		        	:= p_tyUSBoardArrivedData.tyData.sBatchId;

					tyBoardForecastSnd.tyAvl.bForecastId 			    := tyBoardForecastSnd.tyData.sForecastId <> '';
					tyBoardForecastSnd.tyAvl.bTimeUntilAvailable		:= tyBoardForecastSnd.tyData.rTimeUntilAvailable <> 0;
					tyBoardForecastSnd.tyAvl.bBoardId 				    := tyBoardForecastSnd.tyData.sBoardId <> '';
					tyBoardForecastSnd.tyAvl.bBoardIdCreatedBy 	    	:= tyBoardForecastSnd.tyData.sBoardIdCreatedBy <> '';
					tyBoardForecastSnd.tyAvl.bFailedBoard 			    := TRUE;
					tyBoardForecastSnd.tyAvl.bProductTypeId 			:= tyBoardForecastSnd.tyData.sProductTypeId <> '';
					tyBoardForecastSnd.tyAvl.bFlippedBoard 		    	:= TRUE;
					tyBoardForecastSnd.tyAvl.bTopBarcode 			    := tyBoardForecastSnd.tyData.sTopBarcode <> '';
					tyBoardForecastSnd.tyAvl.bBottomBarcode 			:= tyBoardForecastSnd.tyData.sBottomBarcode <> '';
					tyBoardForecastSnd.tyAvl.bLength 				    := tyBoardForecastSnd.tyData.rLength <> 0;
					tyBoardForecastSnd.tyAvl.bWidth 				    := tyBoardForecastSnd.tyData.rWidth <> 0;
					tyBoardForecastSnd.tyAvl.bThickness 			    := tyBoardForecastSnd.tyData.rThickness <> 0;
					tyBoardForecastSnd.tyAvl.bConveyorSpeed 			:= tyBoardForecastSnd.tyData.rConveyorSpeed <> 0;
					tyBoardForecastSnd.tyAvl.bTopClearanceHeight 		:= tyBoardForecastSnd.tyData.rTopClearanceHeight <> 0;
					tyBoardForecastSnd.tyAvl.bBottomClearanceHeight 	:= tyBoardForecastSnd.tyData.rBottomClearanceHeight <> 0;
					tyBoardForecastSnd.tyAvl.bWeight 			    	:= tyBoardForecastSnd.tyData.rWeight <> 0;
					tyBoardForecastSnd.tyAvl.bWorkOrderId 		    	:= tyBoardForecastSnd.tyData.sWorkOrderId <> '';
					tyBoardForecastSnd.tyAvl.bBatchId 		        	:= tyBoardForecastSnd.tyData.sBatchId <> '';

				END_IF
			END_IF

		ELSIF fbSequenceDS.eMsgTypeSnd = HermesMsgTypeBoardAvailable THEN
			fHermesAddOneMsgSend(ADR(a_eMsgSend) , ADR(udiMsgSendBffr) , HermesMsgTypeBoardAvailable);

				IF (p_eLinkCustomerReq = NA OR p_sWorkOrderId = '' OR p_usiProdRcpCurrRcp1McMod = 0) AND p_bNewBrdAvlLastZone = TRUE AND p_bRcvBoardInfo = FALSE THEN //Generate New B.A for Unknown PCB

					fHermesGenerateUUID(ADR(tyBoardAvailableSnd.tyData.sBoardId) , p_tyDTStructure , pa_usiMacAddr);

					tyBoardAvailableSnd.tyData.sBoardIdCreatedBy        := p_sMcId; //Generate by our Machine
					tyBoardAvailableSnd.tyData.eFailedBoard				:= p_eFailedBoard;
					tyBoardAvailableSnd.tyData.sProductTypeId			:= p_sRecipeNm;
					tyBoardAvailableSnd.tyData.eFlippedBoard			:= p_eFlippedBoard;
					tyBoardAvailableSnd.tyData.sTopBarcode				:= p_sTopBarcode;
					tyBoardAvailableSnd.tyData.sBottomBarcode			:= p_sBottomBarcode;
					tyBoardAvailableSnd.tyData.rLength					:= p_rLength;
					tyBoardAvailableSnd.tyData.rWidth					:= DINT_TO_REAL(p_diWidthInUM) / 1000;
					tyBoardAvailableSnd.tyData.rThickness				:= p_rThickness;
					tyBoardAvailableSnd.tyData.rConveyorSpeed			:= p_rConveyorSpeed;
					tyBoardAvailableSnd.tyData.rTopClearanceHeight		:= p_rTopClearanceHeight;
					tyBoardAvailableSnd.tyData.rBottomClearanceHeight	:= p_rBottomClearanceHeight;
					tyBoardAvailableSnd.tyData.rWeight					:= p_rWeight;
//					tyBoardAvailableSnd.tyData.sWorkOrderId			    := p_sWorkOrderId;
//					tyBoardAvailableSnd.tyData.sBatchId			        := p_sBatchId;
					tyBoardAvailableSnd.tyData.sWorkOrderId			    := '';
					tyBoardAvailableSnd.tyData.sBatchId			        := '';

					tyBoardAvailableSnd.tyAvl.bBoardId					:= tyBoardAvailableSnd.tyData.sBoardId<>'';
					tyBoardAvailableSnd.tyAvl.bBoardIdCreatedBy			:= tyBoardAvailableSnd.tyData.sBoardIdCreatedBy <> '';
					tyBoardAvailableSnd.tyAvl.bFailedBoard				:= TRUE;
					tyBoardAvailableSnd.tyAvl.bProductTypeId			:= tyBoardAvailableSnd.tyData.sProductTypeId <> '';
					tyBoardAvailableSnd.tyAvl.bFlippedBoard				:= TRUE;
					tyBoardAvailableSnd.tyAvl.bTopBarcode				:= tyBoardAvailableSnd.tyData.sTopBarcode <> '';
					tyBoardAvailableSnd.tyAvl.bBottomBarcode			:= tyBoardAvailableSnd.tyData.sBottomBarcode <> '';
					tyBoardAvailableSnd.tyAvl.bLength					:= tyBoardAvailableSnd.tyData.rLength <> 0;
					tyBoardAvailableSnd.tyAvl.bWidth					:= (tyBoardAvailableSnd.tyData.rWidth <> 0) AND (p_bBAWidthEn = TRUE);
					tyBoardAvailableSnd.tyAvl.bThickness				:= (tyBoardAvailableSnd.tyData.rThickness <> 0) AND (p_bBASltEn = TRUE);
					tyBoardAvailableSnd.tyAvl.bConveyorSpeed			:= tyBoardAvailableSnd.tyData.rConveyorSpeed <> 0;
					tyBoardAvailableSnd.tyAvl.bTopClearanceHeight		:= (tyBoardAvailableSnd.tyData.rTopClearanceHeight <> 0) AND (p_bBASltEn = TRUE);
					tyBoardAvailableSnd.tyAvl.bBottomClearanceHeight	:= (tyBoardAvailableSnd.tyData.rBottomClearanceHeight <> 0) AND (p_bBASltEn = TRUE);
					tyBoardAvailableSnd.tyAvl.bWeight					:= tyBoardAvailableSnd.tyData.rWeight <> 0;
					tyBoardAvailableSnd.tyAvl.bWorkOrderId				:= tyBoardAvailableSnd.tyData.sWorkOrderId <> '';
					tyBoardAvailableSnd.tyAvl.bBatchId			    	:= tyBoardAvailableSnd.tyData.sBatchId <> '';

				ELSIF p_eLinkCustomerReq = Siemens AND p_sWorkOrderId <>'' AND (p_usiProdRcpCurrRcp1McMod = 1)  AND p_bNewBrdAvlLastZone = TRUE AND p_bRcvBoardInfo = FALSE THEN //Data from Supervisory(Siemens)

					fHermesGenerateUUID(ADR(tyBoardAvailableSnd.tyData.sBoardId) , p_tyDTStructure , pa_usiMacAddr);

					tyBoardAvailableSnd.tyData.sBoardIdCreatedBy        := p_sMcId;
					tyBoardAvailableSnd.tyData.eFailedBoard				:= p_eFailedBoard;
					tyBoardAvailableSnd.tyData.sProductTypeId			:= p_tySendWorkOrderData.tyData.sProductTypeId;
					tyBoardAvailableSnd.tyData.eFlippedBoard			:= p_eFlippedBoard;
					tyBoardAvailableSnd.tyData.sTopBarcode				:= p_sTopBarcode;
					tyBoardAvailableSnd.tyData.sBottomBarcode			:= p_sBottomBarcode;
					tyBoardAvailableSnd.tyData.rLength					:= p_tySendWorkOrderData.tyData.rLength;
					tyBoardAvailableSnd.tyData.rWidth					:= p_tySendWorkOrderData.tyData.rWidth;
					tyBoardAvailableSnd.tyData.rThickness				:= p_tySendWorkOrderData.tyData.rThickness;
					tyBoardAvailableSnd.tyData.rConveyorSpeed			:= p_rConveyorSpeed; //dont have
					tyBoardAvailableSnd.tyData.rTopClearanceHeight		:= p_tySendWorkOrderData.tyData.rTopClearanceHeight;
					tyBoardAvailableSnd.tyData.rBottomClearanceHeight	:= p_tySendWorkOrderData.tyData.rBottomClearanceHeight;
					tyBoardAvailableSnd.tyData.rWeight					:= p_tySendWorkOrderData.tyData.rWeight;
					tyBoardAvailableSnd.tyData.sWorkOrderId			    := p_tySendWorkOrderData.tyData.sWorkOrderId;
					tyBoardAvailableSnd.tyData.sBatchId		            := p_tySendWorkOrderData.tyData.sBatchId;

					tyBoardAvailableSnd.tyAvl.bBoardId					:= tyBoardAvailableSnd.tyData.sBoardId<>'';
					tyBoardAvailableSnd.tyAvl.bBoardIdCreatedBy			:= tyBoardAvailableSnd.tyData.sBoardIdCreatedBy <> '';
					tyBoardAvailableSnd.tyAvl.bFailedBoard				:= TRUE;
					tyBoardAvailableSnd.tyAvl.bProductTypeId			:= tyBoardAvailableSnd.tyData.sProductTypeId <> '';
					tyBoardAvailableSnd.tyAvl.bFlippedBoard				:= TRUE;
					tyBoardAvailableSnd.tyAvl.bTopBarcode				:= tyBoardAvailableSnd.tyData.sTopBarcode <> '';
					tyBoardAvailableSnd.tyAvl.bBottomBarcode			:= tyBoardAvailableSnd.tyData.sBottomBarcode <> '';
					tyBoardAvailableSnd.tyAvl.bLength					:= tyBoardAvailableSnd.tyData.rLength <> 0;
					tyBoardAvailableSnd.tyAvl.bWidth					:= (tyBoardAvailableSnd.tyData.rWidth <> 0) AND (p_bBAWidthEn = TRUE);
					tyBoardAvailableSnd.tyAvl.bThickness				:= (tyBoardAvailableSnd.tyData.rThickness <> 0) AND (p_bBASltEn = TRUE);
					tyBoardAvailableSnd.tyAvl.bConveyorSpeed			:= tyBoardAvailableSnd.tyData.rConveyorSpeed <> 0;
					tyBoardAvailableSnd.tyAvl.bTopClearanceHeight		:= (tyBoardAvailableSnd.tyData.rTopClearanceHeight <> 0) AND (p_bBASltEn = TRUE);
					tyBoardAvailableSnd.tyAvl.bBottomClearanceHeight	:= (tyBoardAvailableSnd.tyData.rBottomClearanceHeight <> 0) AND (p_bBASltEn = TRUE);
					tyBoardAvailableSnd.tyAvl.bWeight					:= tyBoardAvailableSnd.tyData.rWeight <> 0;
					tyBoardAvailableSnd.tyAvl.bWorkOrderId				:= tyBoardAvailableSnd.tyData.sWorkOrderId <> '';
					tyBoardAvailableSnd.tyAvl.bBatchId			    	:= tyBoardAvailableSnd.tyData.sBatchId <> '';

					/////////////////////////////////////////

				ELSIF p_bNewBrdAvlLastZone = TRUE AND p_bRcvBoardInfo = TRUE THEN //Take BoardInfo From "SendBoardInfo", for Manual Insert PCB

					tyBoardAvailableSnd.tyData.sBoardId                 := p_tyBoardInfoData.tyData.sBoardId;
					tyBoardAvailableSnd.tyData.sBoardIdCreatedBy        := p_tyBoardInfoData.tyData.sBoardIdCreatedBy;
					tyBoardAvailableSnd.tyData.eFailedBoard				:= p_tyBoardInfoData.tyData.eFailedBoard;
					tyBoardAvailableSnd.tyData.sProductTypeId			:= p_tyBoardInfoData.tyData.sProductTypeId;
					tyBoardAvailableSnd.tyData.eFlippedBoard			:= p_tyBoardInfoData.tyData.eFlippedBoard;
					tyBoardAvailableSnd.tyData.sTopBarcode				:= p_tyBoardInfoData.tyData.sTopBarcode;
					tyBoardAvailableSnd.tyData.sBottomBarcode			:= p_tyBoardInfoData.tyData.sBottomBarcode;
					tyBoardAvailableSnd.tyData.rLength					:= p_tyBoardInfoData.tyData.rLength;
					tyBoardAvailableSnd.tyData.rWidth					:= p_tyBoardInfoData.tyData.rWidth;
					tyBoardAvailableSnd.tyData.rThickness				:= p_tyBoardInfoData.tyData.rThickness;
					tyBoardAvailableSnd.tyData.rConveyorSpeed			:= p_rConveyorSpeed; //dont have
					tyBoardAvailableSnd.tyData.rTopClearanceHeight		:= p_tyBoardInfoData.tyData.rTopClearanceHeight;
					tyBoardAvailableSnd.tyData.rBottomClearanceHeight	:= p_tyBoardInfoData.tyData.rBottomClearanceHeight;
					tyBoardAvailableSnd.tyData.rWeight					:= p_tyBoardInfoData.tyData.rWeight;
					tyBoardAvailableSnd.tyData.sWorkOrderId			    := p_tyBoardInfoData.tyData.sWorkOrderId;
					tyBoardAvailableSnd.tyData.sBatchId		            := p_tyBoardInfoData.tyData.sBatchId;

					tyBoardAvailableSnd.tyAvl.bBoardId					:= tyBoardAvailableSnd.tyData.sBoardId <> '';
					tyBoardAvailableSnd.tyAvl.bBoardIdCreatedBy			:= tyBoardAvailableSnd.tyData.sBoardIdCreatedBy <> '';
					tyBoardAvailableSnd.tyAvl.bFailedBoard				:= TRUE;
					tyBoardAvailableSnd.tyAvl.bProductTypeId			:= tyBoardAvailableSnd.tyData.sProductTypeId <> '';
					tyBoardAvailableSnd.tyAvl.bFlippedBoard				:= TRUE;
					tyBoardAvailableSnd.tyAvl.bTopBarcode				:= tyBoardAvailableSnd.tyData.sTopBarcode <> '';
					tyBoardAvailableSnd.tyAvl.bBottomBarcode			:= tyBoardAvailableSnd.tyData.sBottomBarcode <> '';
					tyBoardAvailableSnd.tyAvl.bLength					:= tyBoardAvailableSnd.tyData.rLength <> 0;
					tyBoardAvailableSnd.tyAvl.bWidth					:= (tyBoardAvailableSnd.tyData.rWidth <> 0);
					tyBoardAvailableSnd.tyAvl.bThickness				:= (tyBoardAvailableSnd.tyData.rThickness <> 0);
					tyBoardAvailableSnd.tyAvl.bConveyorSpeed			:= tyBoardAvailableSnd.tyData.rConveyorSpeed <> 0;
					tyBoardAvailableSnd.tyAvl.bTopClearanceHeight		:= (tyBoardAvailableSnd.tyData.rTopClearanceHeight <> 0);
					tyBoardAvailableSnd.tyAvl.bBottomClearanceHeight	:= (tyBoardAvailableSnd.tyData.rBottomClearanceHeight <> 0);
			tyBoardAvailableSnd.tyAvl.bWeight					:= tyBoardAvailableSnd.tyData.rWeight <> 0;
			tyBoardAvailableSnd.tyAvl.bWorkOrderId				:= tyBoardAvailableSnd.tyData.sWorkOrderId <> '';
			tyBoardAvailableSnd.tyAvl.bBatchId			    	:= tyBoardAvailableSnd.tyData.sBatchId <> '';

		ELSE //Take from PCB_In Board Data

			fbParseBrdAvlExternal.p_XMLTable		:= ADR(pa_tyXMLTableDataBrdAvl); //last zone B.A
			fbParseBrdAvlExternal.iTotalIdxWrite	:= p_iXMLTableDataBrdAvlTtlIdx; //last zone
			fbParseBrdAvlExternal;
			tyBoardAvailableSnd	:= fbParseBrdAvlExternal.tyBoardAvailable;
		END_IF

	ELSIF fbSequenceDS.eMsgTypeSnd = HermesMsgTypeRevokeBoardAvl THEN
		fHermesAddOneMsgSend(ADR(a_eMsgSend) , ADR(udiMsgSendBffr) , HermesMsgTypeRevokeBoardAvl);

	ELSIF fbSequenceDS.eMsgTypeSnd = HermesMsgTypeTransportFinished THEN
		fHermesAddOneMsgSend(ADR(a_eMsgSend) , ADR(udiMsgSendBffr) , HermesMsgTypeTransportFinished);

		IF p_bSndCompl = TRUE THEN
			tyTransportFinished.tyData.eTransferState	:= HermesTransferStateComplete;
		ELSIF p_bSndIncompl = TRUE THEN
			tyTransportFinished.tyData.eTransferState	:= HermesTransferStateIncomplete;
		ELSE
			tyTransportFinished.tyData.eTransferState	:= HermesTransferStateNotStarted;
		END_IF
		tyTransportFinished.tyData.sBoardId				:= tyStartTransport.tyData.sBoardId;

		tyTransportFinished.tyAvl.bTransferState		:= TRUE;
		tyTransportFinished.tyAvl.bBoardId				:= TRUE;

	END_IF

	END_IF

END_ACTION
```

#### Act_Background_SendBoardInfo.st - Do Not Change!!!
```iecst
(** 2021-08-01 **)
ACTION Act_Background_SendBoardInfo:

	IF eStatus2 <> Error THEN
		IF tyServiceDescriptionRcv.tyAvl.tySupportedFeatures.bFeatureQueryBoardInfo = TRUE AND p_tyParam.bFeatureSendBoardInfo THEN

			IF tyMsgTypeRcv.bQueryBoardInfo THEN

			    IF tyQueryBoardInfo.tyData.sTopBarcode <> '' THEN
					bSearchTop := TRUE;
					sSearchTop := tyQueryBoardInfo.tyData.sTopBarcode;
				ELSE
				    bSearchTop := FALSE;
				END_IF

				IF tyQueryBoardInfo.tyData.sBottomBarcode <> '' THEN
					bSearchBottom := TRUE;
					sSearchBottom := tyQueryBoardInfo.tyData.sBottomBarcode;
				ELSE
					bSearchBottom := FALSE;
				END_IF

				udiTopTargetAddress := ADR(a_tyBoardDepartedInfo[0].tyData.sTopBarcode); //Top Barcode Start address
				udiBottomTargetAddress := ADR(a_tyBoardDepartedInfo[0].tyData.sBottomBarcode); //Bottom Barcode Start address
				udiSizeOfAddress := SIZEOF(a_tyBoardDepartedInfo[0]); //Size of one recipe

				// Search Top Barcode
				IF bSearchTop = TRUE THEN

					FOR j := 0 TO 49 DO //50 recipes

							IF memcmp((udiTopTargetAddress)+(j*udiSizeOfAddress), ADR(sSearchTop) , LEN(sSearchTop)) = 0 THEN

								bFoundTop	:= TRUE;
							    udiFoundRecipeTop := j;
								udiFoundAddressTop := (udiTopTargetAddress)+(j*udiSizeOfAddress);
								p_sFoundAddressTop ACCESS (udiFoundAddressTop);
								EXIT;
							END_IF

					END_FOR
				END_IF

				// Search Bottom Barcode

				IF bSearchBottom = TRUE THEN

					FOR jj := 0 TO 49 DO

							IF memcmp((udiBottomTargetAddress)+(jj*udiSizeOfAddress), ADR(sSearchBottom) , LEN(sSearchBottom)) = 0 THEN

								bFoundBottom	:= TRUE;
							    udiFoundRecipeBottom := jj;
								udiFoundAddressBottom := (udiBottomTargetAddress)+(jj*udiSizeOfAddress);
								p_sFoundAddressBottom ACCESS (udiFoundAddressBottom);
								EXIT;
							END_IF

					END_FOR
				END_IF

				IF bSearchTop AND bSearchBottom AND bFoundTop AND bFoundBottom THEN
					IF udiFoundRecipeTop <> udiFoundRecipeBottom THEN //No need Error
						bSendOk := TRUE;
				    	bFoundNothing := TRUE;
					ELSE
						bSendOk := TRUE;
					    bFoundNothing := FALSE;
					    udiFoundRecipeFinal := udiFoundRecipeTop OR udiFoundRecipeBottom; //Both are same.
					END_IF

				ELSIF bSearchTop AND bSearchBottom AND bFoundTop AND bFoundBottom = FALSE THEN
					bSendOk := TRUE;
					bFoundNothing := TRUE;

				ELSIF bSearchTop AND bSearchBottom AND bFoundTop = FALSE AND bFoundBottom THEN
					bSendOk := TRUE;
					bFoundNothing := TRUE;

				ELSIF bSearchTop AND bSearchBottom AND bFoundTop = FALSE AND bFoundBottom = FALSE THEN
					bSendOk := TRUE;
					bFoundNothing := TRUE;
				END_IF

				IF bSearchTop AND bSearchBottom = FALSE AND bFoundTop THEN
					bSendOk := TRUE;
					bFoundNothing := FALSE;
					udiFoundRecipeFinal := udiFoundRecipeTop;
				END_IF

				IF bSearchTop AND bSearchBottom = FALSE AND bFoundTop = FALSE THEN
					bSendOk := TRUE;
					bFoundNothing := TRUE;
				END_IF

				IF bSearchTop = FALSE AND bSearchBottom AND bFoundBottom THEN
					bSendOk := TRUE;
					bFoundNothing := FALSE;
					udiFoundRecipeFinal := udiFoundRecipeBottom;
				END_IF

				IF bSearchTop = FALSE AND bSearchBottom AND bFoundBottom = FALSE THEN
					bSendOk := TRUE;
					bFoundNothing := TRUE;
				END_IF

				IF  bSendOk AND bFoundNothing = FALSE THEN //BoardInfo Found

					fHermesAddOneMsgSend(ADR(a_eMsgSend) , ADR(udiMsgSendBffr) , HermesMsgTypeSendBoardInfo);

					tySendBoardInfo.tyData.sBoardId                     := a_tyBoardDepartedInfo[udiFoundRecipeFinal].tyData.sBoardId;
					tySendBoardInfo.tyData.sBoardIdCreatedBy            := a_tyBoardDepartedInfo[udiFoundRecipeFinal].tyData.sBoardIdCreatedBy;
					tySendBoardInfo.tyData.eFailedBoard 		    	:= a_tyBoardDepartedInfo[udiFoundRecipeFinal].tyData.eFailedBoard;
					tySendBoardInfo.tyData.sProductTypeId 			    := a_tyBoardDepartedInfo[udiFoundRecipeFinal].tyData.sProductTypeId;	 //current recipe0 name
					tySendBoardInfo.tyData.eFlippedBoard 		    	:= a_tyBoardDepartedInfo[udiFoundRecipeFinal].tyData.eFlippedBoard;
					tySendBoardInfo.tyData.sTopBarcode 		        	:= a_tyBoardDepartedInfo[udiFoundRecipeFinal].tyData.sTopBarcode;
					tySendBoardInfo.tyData.sBottomBarcode 		    	:= a_tyBoardDepartedInfo[udiFoundRecipeFinal].tyData.sBottomBarcode;
					tySendBoardInfo.tyData.rLength 			        	:= a_tyBoardDepartedInfo[udiFoundRecipeFinal].tyData.rLength;
					tySendBoardInfo.tyData.rWidth 			        	:= a_tyBoardDepartedInfo[udiFoundRecipeFinal].tyData.rWidth;	//current recipe 0 width
					tySendBoardInfo.tyData.rThickness 		        	:= a_tyBoardDepartedInfo[udiFoundRecipeFinal].tyData.rThickness;
					tySendBoardInfo.tyData.rTopClearanceHeight 	    	:= a_tyBoardDepartedInfo[udiFoundRecipeFinal].tyData.rTopClearanceHeight;
					tySendBoardInfo.tyData.rBottomClearanceHeight 	    := a_tyBoardDepartedInfo[udiFoundRecipeFinal].tyData.rBottomClearanceHeight;
					tySendBoardInfo.tyData.rWeight 			        	:= a_tyBoardDepartedInfo[udiFoundRecipeFinal].tyData.rWeight;
					tySendBoardInfo.tyData.sWorkOrderId 		    	:= a_tyBoardDepartedInfo[udiFoundRecipeFinal].tyData.sWorkOrderId;

		    		tySendBoardInfo.tyAvl.bBoardId 				        := tySendBoardInfo.tyData.sBoardId <> '';
		    		tySendBoardInfo.tyAvl.bBoardIdCreatedBy 	        := tySendBoardInfo.tyData.sBoardIdCreatedBy <> '';
		    		tySendBoardInfo.tyAvl.bFailedBoard 			        := TRUE;
		    		tySendBoardInfo.tyAvl.bProductTypeId 		    	:= tySendBoardInfo.tyData.sProductTypeId <> '';
		    		tySendBoardInfo.tyAvl.bFlippedBoard 		        := TRUE;
		    		tySendBoardInfo.tyAvl.bTopBarcode 		    	    := tySendBoardInfo.tyData.sTopBarcode <> '';
					tySendBoardInfo.tyAvl.bBottomBarcode 		    	:= tySendBoardInfo.tyData.sBottomBarcode <> '';
					tySendBoardInfo.tyAvl.bWidth 			        	:= tySendBoardInfo.tyData.rWidth <> 0;
		    		tySendBoardInfo.tyAvl.bLength 			        	:= tySendBoardInfo.tyData.rLength <> 0;
		 	    	tySendBoardInfo.tyAvl.bThickness 		        	:= tySendBoardInfo.tyData.rThickness <> 0;
			    	tySendBoardInfo.tyAvl.bTopClearanceHeight 	    	:= tySendBoardInfo.tyData.rTopClearanceHeight <> 0;
			    	tySendBoardInfo.tyAvl.bBottomClearanceHeight 	    := tySendBoardInfo.tyData.rBottomClearanceHeight <> 0;
			    	tySendBoardInfo.tyAvl.bWeight 			        	:= tySendBoardInfo.tyData.rWeight <> 0;
			    	tySendBoardInfo.tyAvl.bWorkOrderId 		        	:= tySendBoardInfo.tyData.sWorkOrderId <> '';

				ELSIF bSendOk AND bFoundNothing = TRUE THEN //BoardInfo Not Found

					fHermesAddOneMsgSend(ADR(a_eMsgSend) , ADR(udiMsgSendBffr) , HermesMsgTypeSendBoardInfo);

					tySendBoardInfo.tyData.sBoardId                     := '';
					tySendBoardInfo.tyData.sBoardIdCreatedBy            := '';
					tySendBoardInfo.tyData.eFailedBoard 		    	:= HermesUnknownBoard;
					tySendBoardInfo.tyData.sProductTypeId 			    := '';
					tySendBoardInfo.tyData.eFlippedBoard 		    	:= HermesFlippedBoardUnknownSide;
					tySendBoardInfo.tyData.sTopBarcode 		        	:= tyQueryBoardInfo.tyData.sTopBarcode;
					tySendBoardInfo.tyData.sBottomBarcode 		    	:= tyQueryBoardInfo.tyData.sBottomBarcode;
					tySendBoardInfo.tyData.rLength 			        	:= 0;
					tySendBoardInfo.tyData.rWidth 			        	:= 0;
					tySendBoardInfo.tyData.rThickness 		        	:= 0;
					tySendBoardInfo.tyData.rTopClearanceHeight 	    	:= 0;
					tySendBoardInfo.tyData.rBottomClearanceHeight 	    := 0;
					tySendBoardInfo.tyData.rWeight 			        	:= 0;
					tySendBoardInfo.tyData.sWorkOrderId 		    	:= '';
					tySendBoardInfo.tyData.sBatchId      		    	:= '';

					tySendBoardInfo.tyAvl.bBoardId 				        := tySendBoardInfo.tyData.sBoardId <> '';
					tySendBoardInfo.tyAvl.bBoardIdCreatedBy 	        := tySendBoardInfo.tyData.sBoardIdCreatedBy <> '';
					tySendBoardInfo.tyAvl.bFailedBoard 			        := FALSE; //no need send
					tySendBoardInfo.tyAvl.bProductTypeId 		    	:= tySendBoardInfo.tyData.sProductTypeId <> '';
					tySendBoardInfo.tyAvl.bFlippedBoard 	    	    := FALSE; //no need send
					tySendBoardInfo.tyAvl.bTopBarcode 		        	:= tySendBoardInfo.tyData.sTopBarcode <> '';
					tySendBoardInfo.tyAvl.bBottomBarcode 	    		:= tySendBoardInfo.tyData.sBottomBarcode <> '';
					tySendBoardInfo.tyAvl.bLength 			        	:= tySendBoardInfo.tyData.rLength <> 0;
					tySendBoardInfo.tyAvl.bWidth 			        	:= tySendBoardInfo.tyData.rWidth <> 0;
					tySendBoardInfo.tyAvl.bThickness 		        	:= tySendBoardInfo.tyData.rThickness <> 0;
					tySendBoardInfo.tyAvl.bTopClearanceHeight 	    	:= tySendBoardInfo.tyData.rTopClearanceHeight <> 0;
					tySendBoardInfo.tyAvl.bBottomClearanceHeight     	:= tySendBoardInfo.tyData.rBottomClearanceHeight <> 0;
					tySendBoardInfo.tyAvl.bWeight 			        	:= tySendBoardInfo.tyData.rWeight <> 0;
					tySendBoardInfo.tyAvl.bWorkOrderId 		        	:= tySendBoardInfo.tyData.sWorkOrderId <> '';
					tySendBoardInfo.tyAvl.bBatchId 		            	:= tySendBoardInfo.tyData.sBatchId <> '';

				END_IF

			ELSE //if tyMsgTypeRcv.bQueryBoardInfo = FALSE
				bFoundTop	   := FALSE;
				bFoundBottom   := FALSE;
				bFoundNothing  := FALSE;
				bSearchTop     := FALSE;
				bSearchBottom  := FALSE;
				bSendOk        := FALSE;
			END_IF

		ELSE //if feature bFeatureQueryBoardInfo not supported
			bFoundTop	   := FALSE;
			bFoundBottom   := FALSE;
			bFoundNothing  := FALSE;
			bSearchTop     := FALSE;
			bSearchBottom  := FALSE;
			bSendOk        := FALSE;
		END_IF
	END_IF

END_ACTION
```

#### Act_Alarm.st - Do Not Change!!!
```iecst
(** 2021-08-01 **)
ACTION Act_Alarm:

	//Error
	IF EDGEPOS(eStatus = Error) THEN

		tyAlmData.sProgNm		:= p_sProgNm;
		tyAlmData.udiCode		:= udiStatus;
		tyAlmData.eSeverity		:= AlmSeverityError;
		tyAlmData.udiRunTime	:= tyAlmData.udiRunTime + 1;
		tyAlmData.bAlm			:= TRUE;
		tyAlmData.udiModuleNum  := udiModuleNum;
		g_sDSHermesBProgNm		:= p_sProgNm;

		//Get Error Message
		IF tyAlmData.udiCode < 10000 OR tyAlmData.udiCode > 10199 THEN
			tyAlmData.sAlmMsg	:= 'Unknown';
			tyAlmData.sRcyMsg	:= 'Unknown';
		ELSE
			tyAlmData.sAlmMsg	:= a_tyAlmText[tyAlmData.udiCode].sAlmText;
			tyAlmData.sRcyMsg	:= a_tyAlmText[tyAlmData.udiCode].sRcyText;
		END_IF

		sStatTxt	:= tyAlmData.sAlmMsg;

	ELSIF bRstErr AND (tyAlmData.udiCode <> 0) THEN

		tyAlmData.udiCode	:= 0;
		tyAlmData.eSeverity	:= AlmSeverityNA;
		tyAlmData.sAlmMsg	:= '';
		tyAlmData.sRcyMsg	:= '';
		tyAlmData.bAlm			:= FALSE;
		sStatTxt	:= a_sStatText[eStat];

	END_IF

END_ACTION
```

#### Act_Alarm1.st - Do Not Change!!!
```iecst
(** 2021-08-01 **)
ACTION Act_Alarm1: //General

	//Error
	IF EDGEPOS(eStatus1 = Error) THEN

		tyAlmData1.sProgNm		:= p_sProgNm;
		tyAlmData1.udiCode		:= udiStatus1;
		tyAlmData1.eSeverity	:= AlmSeverityError;
		tyAlmData1.udiRunTime	:= tyAlmData1.udiRunTime + 1;
		tyAlmData1.bAlm			:= TRUE;
		tyAlmData1.udiModuleNum  := udiModuleNum;
		g_sDSHermesBProgNm		:= p_sProgNm;
		//Get Error Message
		IF tyAlmData1.udiCode < 10000 OR tyAlmData1.udiCode > 10199 THEN
			tyAlmData1.sAlmMsg	:= 'Unknown';
			tyAlmData1.sRcyMsg	:= 'Unknown';
		ELSE
			tyAlmData1.sAlmMsg	:= a_tyAlmText[tyAlmData1.udiCode].sAlmText;
			tyAlmData1.sRcyMsg	:= a_tyAlmText[tyAlmData1.udiCode].sRcyText;
		END_IF

		sStatTxt	:= tyAlmData1.sAlmMsg;

	ELSIF bRstErr AND (tyAlmData1.udiCode <> 0) THEN

		tyAlmData1.udiCode		:= 0;
		tyAlmData1.eSeverity	:= AlmSeverityNA;
		tyAlmData1.sAlmMsg		:= '';
		tyAlmData1.sRcyMsg		:= '';
		tyAlmData1.bAlm			:= FALSE;
		sStatTxt	:= a_sStatText[eStat];

	END_IF

END_ACTION
```

#### Act_Alarm2.st - Do Not Change!!!
```iecst
(** 2019-03-25 **)
ACTION Act_Alarm2:

	//Error
	IF EDGEPOS(eStatus2 = Error) THEN

		tyAlmData2.sProgNm		:= p_sProgNm;
		tyAlmData2.udiCode		:= udiStatus2;
		tyAlmData2.eSeverity	:= AlmSeverityError;
		tyAlmData2.udiRunTime	:= tyAlmData2.udiRunTime + 1;
		tyAlmData2.bAlm			:= TRUE;
		tyAlmData2.udiModuleNum  := udiModuleNum;
		g_sDSHermesBProgNm		:= p_sProgNm;
		//Get Error Message
		IF tyAlmData2.udiCode < 10000 OR tyAlmData2.udiCode > 10199 THEN
			tyAlmData2.sAlmMsg	:= 'Unknown';
			tyAlmData2.sRcyMsg	:= 'Unknown';
		ELSE
			tyAlmData2.sAlmMsg	:= a_tyAlmText[tyAlmData2.udiCode].sAlmText;
			tyAlmData2.sRcyMsg	:= a_tyAlmText[tyAlmData2.udiCode].sRcyText;
		END_IF

		sStatTxt	:= tyAlmData2.sAlmMsg;

	ELSIF bRstErr AND (tyAlmData2.udiCode <> 0) THEN

		tyAlmData2.udiCode		:= 0;
		tyAlmData2.eSeverity	:= AlmSeverityNA;
		tyAlmData2.sAlmMsg		:= '';
		tyAlmData2.sRcyMsg		:= '';
		tyAlmData2.bAlm			:= FALSE;
		sStatTxt	:= a_sStatText[eStat];

	END_IF

END_ACTION
```

#### Act_Alarm3.st - Do Not Change!!!
```iecst
(** 2021-08-01 **)
ACTION Act_Alarm3: //fbFileAppend1 Error

	//Error
	IF EDGEPOS(eStatus3 = Error) THEN

		tyAlmData3.sProgNm		:= p_sProgNm;
		tyAlmData3.udiCode		:= udiStatus3;
		tyAlmData3.eSeverity	:= AlmSeverityError;
		tyAlmData3.udiRunTime	:= tyAlmData3.udiRunTime + 1;
		tyAlmData3.bAlm			:= TRUE;
		tyAlmData3.udiModuleNum  := udiModuleNum;
		g_sDSHermesBProgNm		:= p_sProgNm;
		//Get Error Message
		IF tyAlmData3.udiCode < 10000 OR tyAlmData3.udiCode > 10199 THEN
			tyAlmData3.sAlmMsg	:= 'Unknown';
			tyAlmData3.sRcyMsg	:= 'Unknown';
		ELSE
			tyAlmData3.sAlmMsg	:= a_tyAlmText[tyAlmData3.udiCode].sAlmText;
			tyAlmData3.sRcyMsg	:= a_tyAlmText[tyAlmData3.udiCode].sRcyText;
		END_IF

		sStatTxt	:= tyAlmData3.sAlmMsg;

	ELSIF bRstErr AND (tyAlmData3.udiCode <> 0) THEN

		tyAlmData3.udiCode		:= 0;
		tyAlmData3.eSeverity	:= AlmSeverityNA;
		tyAlmData3.sAlmMsg		:= '';
		tyAlmData3.sRcyMsg		:= '';
		tyAlmData3.bAlm			:= FALSE;
		sStatTxt	:= a_sStatText[eStat];

	END_IF

END_ACTION
```

#### Act_Alarm4.st - Do Not Change!!!
```iecst
(** 2021-08-01 **)
ACTION Act_Alarm4: //Not Connected Warning

	//Warning
	IF ((bConnected = FALSE) AND (p_eLinkMcParamDSCommMod= McSetCommModHermes)) THEN

		tyAlmData4.sProgNm		:= p_sProgNm;
		tyAlmData4.udiCode		:= udiStatus4;
		tyAlmData4.eSeverity	:= AlmSeverityWarning;
		tyAlmData4.udiRunTime	:= tyAlmData4.udiRunTime + 1;
		tyAlmData4.bWarning			:= TRUE;
		tyAlmData4.udiModuleNum  := udiModuleNum;
		g_sDSHermesBProgNm		:= p_sProgNm;
		//Get Error Message
		IF tyAlmData4.udiCode < 10000 OR tyAlmData4.udiCode > 10199 THEN
			tyAlmData4.sAlmMsg	:= 'Unknown';
			tyAlmData4.sRcyMsg	:= 'Unknown';
		ELSE
			tyAlmData4.sAlmMsg	:= a_tyAlmText[tyAlmData4.udiCode].sAlmText;
			tyAlmData4.sRcyMsg	:= a_tyAlmText[tyAlmData4.udiCode].sRcyText;
		END_IF

		sStatTxt	:= tyAlmData4.sAlmMsg;

	ELSIF (bConnected AND (tyAlmData4.udiCode <> 0)) OR (p_eLinkMcParamDSCommMod= McSetCommModSMEMA) THEN

		tyAlmData4.udiCode		:= 0;
		tyAlmData4.eSeverity	:= AlmSeverityNA;
		tyAlmData4.sAlmMsg		:= '';
		tyAlmData4.sRcyMsg		:= '';
		tyAlmData4.bWarning			:= FALSE;
		sStatTxt	:= a_sStatText[eStat];

	END_IF

END_ACTION
```
